   1:L PR[91] R[100]mm/sec CNT100;
   1:  PR[91,1] = PR[90,1] + 41.639;
   1:  PR[91,2] = PR[90,2] + -7.511;
   1:L PR[91] R[100]mm/sec CNT100;
   1:  PR[91,1] = PR[90,1] + 42.015;
   1:  PR[91,2] = PR[90,2] + -6.602;
   1:L PR[91] R[100]mm/sec CNT100;
   1:  PR[91,1] = PR[90,1] + 42.645;
   1:  PR[91,2] = PR[90,2] + -4.250;
   1:L PR[91] R[100]mm/sec CNT100;
   1:  PR[91,1] = PR[90,1] + 42.870;
   1:  PR[91,2] = PR[90,2] + -1.671;
   1:L PR[91] R[100]mm/sec CNT100;
   1:  PR[91,1] = PR[90,1] + 42.984;
   1:  PR[91,2] = PR[90,2] + -0.700;
   1:L PR[91] R[100]mm/sec CNT100;
   1:  PR[91,1] = PR[90,1] + 42.778;
   1:  PR[91,2] = PR[90,2] + 1.658;
   1:L PR[91] R[100]mm/sec CNT100;
   1:  PR[91,1] = PR[90,1] + 42.775;
   1:  PR[91,2] = PR[90,2] + 1.848;
   1:L PR[91] R[100]mm/sec CNT100;
   1:  PR[91,1] = PR[90,1] + 42.656;
   1:  PR[91,2] = PR[90,2] + 2.749;
   1:L PR[91] R[100]mm/sec CNT100;
   1:  PR[91,1] = PR[90,1] + 42.015;
   1:  PR[91,2] = PR[90,2] + 5.145;
   1:L PR[91] R[100]mm/sec CNT100;
   1:  PR[91,1] = PR[90,1] + 41.639;
   1:  PR[91,2] = PR[90,2] + 6.053;
   1:L PR[91] R[100]mm/sec CNT100;
   1:  PR[91,1] = PR[90,1] + 40.576;
   1:  PR[91,2] = PR[90,2] + 8.332;
   1:L PR[91] R[100]mm/sec CNT100;
   1:  PR[91,1] = PR[90,1] + 39.128;
   1:  PR[91,2] = PR[90,2] + 10.399;
   1:L PR[91] R[100]mm/sec CNT100;
   1:  PR[91,1] = PR[90,1] + 38.528;
   1:  PR[91,2] = PR[90,2] + 11.183;
   1:L PR[91] R[100]mm/sec CNT100;
   1:  PR[91,1] = PR[90,1] + 36.785;
   1:  PR[91,2] = PR[90,2] + 12.925;
   1:L PR[91] R[100]mm/sec CNT100;
   1:  PR[91,1] = PR[90,1] + 35.993;
   1:  PR[91,2] = PR[90,2] + 13.534;
   1:L PR[91] R[100]mm/sec CNT100;
   1:  PR[91,1] = PR[90,1] + 33.939;
   1:  PR[91,2] = PR[90,2] + 14.971;
   1:L PR[91] R[100]mm/sec CNT100;
   1:  PR[91,1] = PR[90,1] + 31.670;
   1:  PR[91,2] = PR[90,2] + 16.028;
   1:L PR[91] R[100]mm/sec CNT100;
   1:  PR[91,1] = PR[90,1] + 30.740;
   1:  PR[91,2] = PR[90,2] + 16.415;
   1:L PR[91] R[100]mm/sec CNT100;
   1:  PR[91,1] = PR[90,1] + 28.367;
   1:  PR[91,2] = PR[90,2] + 17.050;
   1:L PR[91] R[100]mm/sec CNT100;
   1:  PR[91,1] = PR[90,1] + 27.353;
   1:  PR[91,2] = PR[90,2] + 17.186;
   1:L PR[91] R[100]mm/sec CNT100;
   1:  PR[91,1] = PR[90,1] + 24.877;
   1:  PR[91,2] = PR[90,2] + 17.401;
   1:L PR[91] R[100]mm/sec CNT100;
   1:  PR[91,1] = PR[90,1] + 22.397;
   1:  PR[91,2] = PR[90,2] + 17.184;
   1:L PR[91] R[100]mm/sec CNT100;
   1:  PR[91,1] = PR[90,1] + 21.373;
   1:  PR[91,2] = PR[90,2] + 17.050;
   1:L PR[91] R[100]mm/sec CNT100;
   1:  PR[91,1] = PR[90,1] + 19.063;
   1:  PR[91,2] = PR[90,2] + 16.431;
   1:L PR[91] R[100]mm/sec CNT100TB   .50sec,CALL END_PUD;
   1:  PR[92] = PR[91];
   1:  PR[92,3] = PR[92,3] + 20;
   1:J PR[92] 10% FINE;
   1:  PR[91,1] = PR[90,1] + 64.674;
   1:  PR[91,2] = PR[90,2] + 14.280;
   1:  PR[92] = PR[91];
   1:  PR[92,3] = PR[92,3] + 20;
   1:J PR[92] 10% FINE;
   1:L PR[91] R[100]mm/sec CNT100;
   1:  CALL LASER_DRAHT_START;
   1:  PR[91,1] = PR[90,1] + 63.262;
   1:  PR[91,2] = PR[90,2] + 13.292;
   1:L PR[91] R[100]mm/sec CNT100;
   1:  PR[91,1] = PR[90,1] + 60.701;
   1:  PR[91,2] = PR[90,2] + 10.743;
   1:L PR[91] R[100]mm/sec CNT100;
   1:  PR[91,1] = PR[90,1] + 59.758;
   1:  PR[91,2] = PR[90,2] + 9.397;
   1:L PR[91] R[100]mm/sec CNT100;
   1:  PR[91,1] = PR[90,1] + 58.704;
   1:  PR[91,2] = PR[90,2] + 7.731;
   1:L PR[91] R[100]mm/sec CNT100;
   1:  PR[91,1] = PR[90,1] + 58.042;
   1:  PR[91,2] = PR[90,2] + 6.310;
   1:L PR[91] R[100]mm/sec CNT100;
   1:  PR[91,1] = PR[90,1] + 57.357;
   1:  PR[91,2] = PR[90,2] + 4.363;
   1:L PR[91] R[100]mm/sec CNT100;
   1:  PR[91,1] = PR[90,1] + 56.969;
   1:  PR[91,2] = PR[90,2] + 2.914;
   1:L PR[91] R[100]mm/sec CNT100;
   1:  PR[91,1] = PR[90,1] + 56.830;
   1:  PR[91,2] = PR[90,2] + 1.324;
   1:L PR[91] R[100]mm/sec CNT100;
   1:  PR[91,1] = PR[90,1] + 56.595;
   1:  PR[91,2] = PR[90,2] + -0.755;
   1:L PR[91] R[100]mm/sec CNT100;
   1:  PR[91,1] = PR[90,1] + 56.725;
   1:  PR[91,2] = PR[90,2] + -2.242;
   1:L PR[91] R[100]mm/sec CNT100;
   1:  PR[91,1] = PR[90,1] + 56.962;
   1:  PR[91,2] = PR[90,2] + -4.348;
   1:L PR[91] R[100]mm/sec CNT100;
   1:  PR[91,1] = PR[90,1] + 57.356;
   1:  PR[91,2] = PR[90,2] + -5.821;
   1:L PR[91] R[100]mm/sec CNT100;
   1:  PR[91,1] = PR[90,1] + 58.041;
   1:  PR[91,2] = PR[90,2] + -7.768;
   1:L PR[91] R[100]mm/sec CNT100;
   1:  PR[91,1] = PR[90,1] + 58.703;
   1:  PR[91,2] = PR[90,2] + -9.188;
   1:L PR[91] R[100]mm/sec CNT100;
   1:  PR[91,1] = PR[90,1] + 59.757;
   1:  PR[91,2] = PR[90,2] + -10.854;
   1:L PR[91] R[100]mm/sec CNT100;
   1:  PR[91,1] = PR[90,1] + 60.699;
   1:  PR[91,2] = PR[90,2] + -12.200;
   1:L PR[91] R[100]mm/sec CNT100;
   1:  PR[91,1] = PR[90,1] + 63.259;
   1:  PR[91,2] = PR[90,2] + -14.749;
   1:L PR[91] R[100]mm/sec CNT100;
   1:  PR[91,1] = PR[90,1] + 64.671;
   1:  PR[91,2] = PR[90,2] + -15.737;
   1:L PR[91] R[100]mm/sec CNT100;
   1:  PR[91,1] = PR[90,1] + 66.191;
   1:  PR[91,2] = PR[90,2] + -16.684;
   1:L PR[91] R[100]mm/sec CNT100;
   1:  PR[91,1] = PR[90,1] + 67.830;
   1:  PR[91,2] = PR[90,2] + -17.448;
   1:L PR[91] R[100]mm/sec CNT100;
   1:  PR[91,1] = PR[90,1] + 69.388;
   1:  PR[91,2] = PR[90,2] + -17.986;
   1:L PR[91] R[100]mm/sec CNT100;
   1:  PR[91,1] = PR[90,1] + 71.205;
   1:  PR[91,2] = PR[90,2] + -18.473;
   1:L PR[91] R[100]mm/sec CNT100;
   1:  PR[91,1] = PR[90,1] + 73.166;
   1:  PR[91,2] = PR[90,2] + -18.646;
   1:L PR[91] R[100]mm/sec CNT100;
   1:  PR[91,1] = PR[90,1] + 74.752;
   1:  PR[91,2] = PR[90,2] + -18.816;
   1:L PR[91] R[100]mm/sec CNT100;
   1:  PR[91,1] = PR[90,1] + 76.727;
   1:  PR[91,2] = PR[90,2] + -18.644;
   1:L PR[91] R[100]mm/sec CNT100;
   1:  PR[91,1] = PR[90,1] + 78.184;
   1:  PR[91,2] = PR[90,2] + -18.473;
   1:L PR[91] R[100]mm/sec CNT100;
   1:  PR[91,1] = PR[90,1] + 80.174;
   1:  PR[91,2] = PR[90,2] + -17.941;
   1:L PR[91] R[100]mm/sec CNT100;
   1:  PR[91,1] = PR[90,1] + 81.453;
   1:  PR[91,2] = PR[90,2] + -17.489;
   1:L PR[91] R[100]mm/sec CNT100;
   1:  PR[91,1] = PR[90,1] + 83.371;
   1:  PR[91,2] = PR[90,2] + -16.595;
   1:L PR[91] R[100]mm/sec CNT100;
   1:  PR[91,1] = PR[90,1] + 84.442;
   1:  PR[91,2] = PR[90,2] + -15.917;
   1:L PR[91] R[100]mm/sec CNT100;
   1:  PR[91,1] = PR[90,1] + 86.225;
   1:  PR[91,2] = PR[90,2] + -14.670;
   1:L PR[91] R[100]mm/sec CNT100;
   1:  PR[91,1] = PR[90,1] + 87.789;
   1:  PR[91,2] = PR[90,2] + -13.107;
   1:L PR[91] R[100]mm/sec CNT100;
   1:  PR[91,1] = PR[90,1] + 88.663;
   1:  PR[91,2] = PR[90,2] + -12.228;
   1:L PR[91] R[100]mm/sec CNT100;
   1:  PR[91,1] = PR[90,1] + 89.933;
   1:  PR[91,2] = PR[90,2] + -10.414;
   1:L PR[91] R[100]mm/sec CNT100;
   1:  PR[91,1] = PR[90,1] + 90.561;
   1:  PR[91,2] = PR[90,2] + -9.412;
   1:L PR[91] R[100]mm/sec CNT100;
   1:  PR[91,1] = PR[90,1] + 91.506;
   1:  PR[91,2] = PR[90,2] + -7.386;
   1:L PR[91] R[100]mm/sec CNT100;
   1:  PR[91,1] = PR[90,1] + 91.883;
   1:  PR[91,2] = PR[90,2] + -6.304;
   1:L PR[91] R[100]mm/sec CNT100;
   1:  PR[91,1] = PR[90,1] + 92.460;
   1:  PR[91,2] = PR[90,2] + -4.148;
   1:L PR[91] R[100]mm/sec CNT100;
   1:  PR[91,1] = PR[90,1] + 92.662;
   1:  PR[91,2] = PR[90,2] + -1.835;
   1:L PR[91] R[100]mm/sec CNT100;
   1:  PR[91,1] = PR[90,1] + 92.788;
   1:  PR[91,2] = PR[90,2] + -0.706;
   1:L PR[91] R[100]mm/sec CNT100;
   1:  PR[91,1] = PR[90,1] + 92.590;
   1:  PR[91,2] = PR[90,2] + 1.557;
   1:L PR[91] R[100]mm/sec CNT100;
   1:  PR[91,1] = PR[90,1] + 92.466;
   1:  PR[91,2] = PR[90,2] + 2.666;
   1:L PR[91] R[100]mm/sec CNT100;
   1:  PR[91,1] = PR[90,1] + 91.883;
   1:  PR[91,2] = PR[90,2] + 4.844;
   1:L PR[91] R[100]mm/sec CNT100;
   1:  PR[91,1] = PR[90,1] + 91.506;
   1:  PR[91,2] = PR[90,2] + 5.927;
   1:L PR[91] R[100]mm/sec CNT100;
   1:  PR[91,1] = PR[90,1] + 90.562;
   1:  PR[91,2] = PR[90,2] + 7.951;
   1:L PR[91] R[100]mm/sec CNT100;
   1:  PR[91,1] = PR[90,1] + 89.935;
   1:  PR[91,2] = PR[90,2] + 8.953;
   1:L PR[91] R[100]mm/sec CNT100;
   1:  PR[91,1] = PR[90,1] + 88.666;
   1:  PR[91,2] = PR[90,2] + 10.765;
   1:L PR[91] R[100]mm/sec CNT100;
   1:  PR[91,1] = PR[90,1] + 86.227;
   1:  PR[91,2] = PR[90,2] + 13.209;
   1:L PR[91] R[100]mm/sec CNT100;
   1:  PR[91,1] = PR[90,1] + 84.447;
   1:  PR[91,2] = PR[90,2] + 14.456;
   1:L PR[91] R[100]mm/sec CNT100;
   1:  PR[91,1] = PR[90,1] + 83.376;
   1:  PR[91,2] = PR[90,2] + 15.134;
   1:L PR[91] R[100]mm/sec CNT100;
   1:  PR[91,1] = PR[90,1] + 81.460;
   1:  PR[91,2] = PR[90,2] + 16.027;
   1:L PR[91] R[100]mm/sec CNT100;
   1:  PR[91,1] = PR[90,1] + 80.180;
   1:  PR[91,2] = PR[90,2] + 16.480;
   1:L PR[91] R[100]mm/sec CNT100;
   1:  PR[91,1] = PR[90,1] + 78.221;
   1:  PR[91,2] = PR[90,2] + 17.005;
   1:L PR[91] R[100]mm/sec CNT100;
   1:  PR[91,1] = PR[90,1] + 76.094;
   1:  PR[91,2] = PR[90,2] + 17.192;
   1:L PR[91] R[100]mm/sec CNT100;
   1:  PR[91,1] = PR[90,1] + 74.710;
   1:  PR[91,2] = PR[90,2] + 17.356;
   1:L PR[91] R[100]mm/sec CNT100;
   1:  PR[91,1] = PR[90,1] + 72.737;
   1:  PR[91,2] = PR[90,2] + 17.184;
   1:L PR[91] R[100]mm/sec CNT100;
   1:  PR[91,1] = PR[90,1] + 71.232;
   1:  PR[91,2] = PR[90,2] + 17.021;
   1:L PR[91] R[100]mm/sec CNT100;
   1:  PR[91,1] = PR[90,1] + 69.394;
   1:  PR[91,2] = PR[90,2] + 16.530;
   1:L PR[91] R[100]mm/sec CNT100;
   1:  PR[91,1] = PR[90,1] + 67.835;
   1:  PR[91,2] = PR[90,2] + 15.992;
   1:L PR[91] R[100]mm/sec CNT100;
   1:  PR[91,1] = PR[90,1] + 66.195;
   1:  PR[91,2] = PR[90,2] + 15.227;
   1:L PR[91] R[100]mm/sec CNT100;
   1:  PR[91,1] = PR[90,1] + 64.674;
   1:  PR[91,2] = PR[90,2] + 14.280;
   1:L PR[91] R[100]mm/sec CNT100TB   .50sec,CALL END_PUD;
   1:  PR[92] = PR[91];
   1:  PR[92,3] = PR[92,3] + 20;
   1:J PR[92] 10% FINE;
   1:  PR[91,1] = PR[90,1] + -7.150;
   1:  PR[91,2] = PR[90,2] + 2.703;
   1:  PR[92] = PR[91];
   1:  PR[92,3] = PR[92,3] + 20;
   1:J PR[92] 10% FINE;
   1:L PR[91] R[100]mm/sec CNT100;
   1:  CALL LASER_DRAHT_START;
   1:  PR[91,1] = PR[90,1] + -7.705;
   1:  PR[91,2] = PR[90,2] + 4.775;
   1:L PR[91] R[100]mm/sec CNT100;
   1:  PR[91,1] = PR[90,1] + -8.126;
   1:  PR[91,2] = PR[90,2] + 5.975;
   1:L PR[91] R[100]mm/sec CNT100;
   1:  PR[91,1] = PR[90,1] + -9.039;
   1:  PR[91,2] = PR[90,2] + 7.935;
   1:L PR[91] R[100]mm/sec CNT100;
   1:  PR[91,1] = PR[90,1] + -9.701;
   1:  PR[91,2] = PR[90,2] + 8.983;
   1:L PR[91] R[100]mm/sec CNT100;
   1:  PR[91,1] = PR[90,1] + -10.954;
   1:  PR[91,2] = PR[90,2] + 10.774;
   1:L PR[91] R[100]mm/sec CNT100;
   1:  PR[91,1] = PR[90,1] + -13.403;
   1:  PR[91,2] = PR[90,2] + 13.218;
   1:L PR[91] R[100]mm/sec CNT100;
   1:  PR[91,1] = PR[90,1] + -15.216;
   1:  PR[91,2] = PR[90,2] + 14.488;
   1:L PR[91] R[100]mm/sec CNT100;
   1:  PR[91,1] = PR[90,1] + -16.211;
   1:  PR[91,2] = PR[90,2] + 15.110;
   1:L PR[91] R[100]mm/sec CNT100;
   1:  PR[91,1] = PR[90,1] + -18.252;
   1:  PR[91,2] = PR[90,2] + 16.062;
   1:L PR[91] R[100]mm/sec CNT100;
   1:  PR[91,1] = PR[90,1] + -19.306;
   1:  PR[91,2] = PR[90,2] + 16.427;
   1:L PR[91] R[100]mm/sec CNT100;
   1:  PR[91,1] = PR[90,1] + -21.495;
   1:  PR[91,2] = PR[90,2] + 17.014;
   1:L PR[91] R[100]mm/sec CNT100;
   1:  PR[91,1] = PR[90,1] + -23.847;
   1:  PR[91,2] = PR[90,2] + 17.220;
   1:L PR[91] R[100]mm/sec CNT100;
   1:  PR[91,1] = PR[90,1] + -24.934;
   1:  PR[91,2] = PR[90,2] + 17.339;
   1:L PR[91] R[100]mm/sec CNT100;
   1:  PR[91,1] = PR[90,1] + -27.250;
   1:  PR[91,2] = PR[90,2] + 17.136;
   1:L PR[91] R[100]mm/sec CNT100;
   1:  PR[91,1] = PR[90,1] + -28.281;
   1:  PR[91,2] = PR[90,2] + 17.016;
   1:L PR[91] R[100]mm/sec CNT100;
   1:  PR[91,1] = PR[90,1] + -30.558;
   1:  PR[91,2] = PR[90,2] + 16.406;
   1:L PR[91] R[100]mm/sec CNT100;
   1:  PR[91,1] = PR[90,1] + -31.489;
   1:  PR[91,2] = PR[90,2] + 16.077;
   1:L PR[91] R[100]mm/sec CNT100;
   1:  PR[91,1] = PR[90,1] + -33.652;
   1:  PR[91,2] = PR[90,2] + 15.068;
   1:L PR[91] R[100]mm/sec CNT100;
   1:  PR[91,1] = PR[90,1] + -34.450;
   1:  PR[91,2] = PR[90,2] + 14.564;
   1:L PR[91] R[100]mm/sec CNT100;
   1:  PR[91,1] = PR[90,1] + -36.424;
   1:  PR[91,2] = PR[90,2] + 13.181;
   1:L PR[91] R[100]mm/sec CNT100;
   1:  PR[91,1] = PR[90,1] + -38.821;
   1:  PR[91,2] = PR[90,2] + 10.781;
   1:L PR[91] R[100]mm/sec CNT100;
   1:  PR[91,1] = PR[90,1] + -40.213;
   1:  PR[91,2] = PR[90,2] + 8.792;
   1:L PR[91] R[100]mm/sec CNT100;
   1:  PR[91,1] = PR[90,1] + -40.692;
   1:  PR[91,2] = PR[90,2] + 8.028;
   1:L PR[91] R[100]mm/sec CNT100;
   1:  PR[91,1] = PR[90,1] + -41.725;
   1:  PR[91,2] = PR[90,2] + 5.811;
   1:L PR[91] R[100]mm/sec CNT100;
   1:  PR[91,1] = PR[90,1] + -42.016;
   1:  PR[91,2] = PR[90,2] + 4.978;
   1:L PR[91] R[100]mm/sec CNT100;
   1:  PR[91,1] = PR[90,1] + -42.644;
   1:  PR[91,2] = PR[90,2] + 2.633;
   1:L PR[91] R[100]mm/sec CNT100;
   1:  PR[91,1] = PR[90,1] + -42.864;
   1:  PR[91,2] = PR[90,2] + 0.118;
   1:L PR[91] R[100]mm/sec CNT100;
   1:  PR[91,1] = PR[90,1] + -42.962;
   1:  PR[91,2] = PR[90,2] + -0.754;
   1:L PR[91] R[100]mm/sec CNT100;
   1:  PR[91,1] = PR[90,1] + -42.748;
   1:  PR[91,2] = PR[90,2] + -3.198;
   1:L PR[91] R[100]mm/sec CNT100;
   1:  PR[91,1] = PR[90,1] + -42.650;
   1:  PR[91,2] = PR[90,2] + -4.066;
   1:L PR[91] R[100]mm/sec CNT100;
   1:  PR[91,1] = PR[90,1] + -42.016;
   1:  PR[91,2] = PR[90,2] + -6.436;
   1:L PR[91] R[100]mm/sec CNT100;
   1:  PR[91,1] = PR[90,1] + -41.725;
   1:  PR[91,2] = PR[90,2] + -7.269;
   1:L PR[91] R[100]mm/sec CNT100;
   1:  PR[91,1] = PR[90,1] + -40.692;
   1:  PR[91,2] = PR[90,2] + -9.486;
   1:L PR[91] R[100]mm/sec CNT100;
   1:  PR[91,1] = PR[90,1] + -40.214;
   1:  PR[91,2] = PR[90,2] + -10.250;
   1:L PR[91] R[100]mm/sec CNT100;
   1:  PR[91,1] = PR[90,1] + -38.822;
   1:  PR[91,2] = PR[90,2] + -12.239;
   1:L PR[91] R[100]mm/sec CNT100;
   1:  PR[91,1] = PR[90,1] + -36.425;
   1:  PR[91,2] = PR[90,2] + -14.639;
   1:L PR[91] R[100]mm/sec CNT100;
   1:  PR[91,1] = PR[90,1] + -34.451;
   1:  PR[91,2] = PR[90,2] + -16.022;
   1:L PR[91] R[100]mm/sec CNT100;
   1:  PR[91,1] = PR[90,1] + -33.653;
   1:  PR[91,2] = PR[90,2] + -16.527;
   1:L PR[91] R[100]mm/sec CNT100;
   1:  PR[91,1] = PR[90,1] + -31.490;
   1:  PR[91,2] = PR[90,2] + -17.536;
   1:L PR[91] R[100]mm/sec CNT100;
   1:  PR[91,1] = PR[90,1] + -30.559;
   1:  PR[91,2] = PR[90,2] + -17.864;
   1:L PR[91] R[100]mm/sec CNT100;
   1:  PR[91,1] = PR[90,1] + -28.309;
   1:  PR[91,2] = PR[90,2] + -18.467;
   1:L PR[91] R[100]mm/sec CNT100;
   1:  PR[91,1] = PR[90,1] + -25.882;
   1:  PR[91,2] = PR[90,2] + -18.680;
   1:L PR[91] R[100]mm/sec CNT100;
   1:  PR[91,1] = PR[90,1] + -24.884;
   1:  PR[91,2] = PR[90,2] + -18.797;
   1:L PR[91] R[100]mm/sec CNT100;
   1:  PR[91,1] = PR[90,1] + -22.569;
   1:  PR[91,2] = PR[90,2] + -18.594;
   1:L PR[91] R[100]mm/sec CNT100;
   1:  PR[91,1] = PR[90,1] + -21.517;
   1:  PR[91,2] = PR[90,2] + -18.479;
   1:L PR[91] R[100]mm/sec CNT100;
   1:  PR[91,1] = PR[90,1] + -19.307;
   1:  PR[91,2] = PR[90,2] + -17.886;
   1:L PR[91] R[100]mm/sec CNT100;
   1:  PR[91,1] = PR[90,1] + -18.253;
   1:  PR[91,2] = PR[90,2] + -17.521;
   1:L PR[91] R[100]mm/sec CNT100;
   1:  PR[91,1] = PR[90,1] + -16.212;
   1:  PR[91,2] = PR[90,2] + -16.569;
   1:L PR[91] R[100]mm/sec CNT100;
   1:  PR[91,1] = PR[90,1] + -15.217;
   1:  PR[91,2] = PR[90,2] + -15.948;
   1:L PR[91] R[100]mm/sec CNT100;
   1:  PR[91,1] = PR[90,1] + -13.404;
   1:  PR[91,2] = PR[90,2] + -14.678;
   1:L PR[91] R[100]mm/sec CNT100;
   1:  PR[91,1] = PR[90,1] + -10.955;
   1:  PR[91,2] = PR[90,2] + -12.233;
   1:L PR[91] R[100]mm/sec CNT100;
   1:  PR[91,1] = PR[90,1] + -9.702;
   1:  PR[91,2] = PR[90,2] + -10.443;
   1:L PR[91] R[100]mm/sec CNT100;
   1:  PR[91,1] = PR[90,1] + -9.040;
   1:  PR[91,2] = PR[90,2] + -9.394;
   1:L PR[91] R[100]mm/sec CNT100;
   1:  PR[91,1] = PR[90,1] + -8.127;
   1:  PR[91,2] = PR[90,2] + -7.435;
   1:L PR[91] R[100]mm/sec CNT100;
   1:  PR[91,1] = PR[90,1] + -7.705;
   1:  PR[91,2] = PR[90,2] + -6.234;
   1:L PR[91] R[100]mm/sec CNT100;
   1:  PR[91,1] = PR[90,1] + -7.157;
   1:  PR[91,2] = PR[90,2] + -4.187;
   1:L PR[91] R[100]mm/sec CNT100;
   1:  PR[91,1] = PR[90,1] + -6.965;
   1:  PR[91,2] = PR[90,2] + -1.986;
   1:L PR[91] R[100]mm/sec CNT100;
   1:  PR[91,1] = PR[90,1] + -6.832;
   1:  PR[91,2] = PR[90,2] + -0.713;
   1:L PR[91] R[100]mm/sec CNT100;
   1:  PR[91,1] = PR[90,1] + -7.035;
   1:  PR[91,2] = PR[90,2] + 1.604;
   1:L PR[91] R[100]mm/sec CNT100;
   1:  PR[91,1] = PR[90,1] + -7.030;
   1:  PR[91,2] = PR[90,2] + 1.640;
   1:L PR[91] R[100]mm/sec CNT100;
   1:  PR[91,1] = PR[90,1] + -7.150;
   1:  PR[91,2] = PR[90,2] + 2.703;
   1:L PR[91] R[100]mm/sec CNT100TB   .50sec,CALL END_PUD;
   1:  PR[92] = PR[91];
   1:  PR[92,3] = PR[92,3] + 20;
   1:J PR[92] 10% FINE;
   1:  PR[91,1] = PR[90,1] + -92.606;
   1:  PR[91,2] = PR[90,2] + 2.602;
   1:  PR[92] = PR[91];
   1:  PR[92,3] = PR[92,3] + 20;
   1:J PR[92] 10% FINE;
   1:L PR[91] R[100]mm/sec CNT100;
   1:  CALL LASER_DRAHT_START;
   1:  PR[91,1] = PR[90,1] + -92.805;
   1:  PR[91,2] = PR[90,2] + 0.315;
   1:L PR[91] R[100]mm/sec CNT100;
   1:  PR[91,1] = PR[90,1] + -92.917;
   1:  PR[91,2] = PR[90,2] + -0.747;
   1:L PR[91] R[100]mm/sec CNT100;
   1:  PR[91,1] = PR[90,1] + -92.733;
   1:  PR[91,2] = PR[90,2] + -2.852;
   1:L PR[91] R[100]mm/sec CNT100;
   1:  PR[91,1] = PR[90,1] + -92.712;
   1:  PR[91,2] = PR[90,2] + -2.937;
   1:L PR[91] R[100]mm/sec CNT100;
   1:  PR[91,1] = PR[90,1] + -92.598;
   1:  PR[91,2] = PR[90,2] + -4.024;
   1:L PR[91] R[100]mm/sec CNT100;
   1:  PR[91,1] = PR[90,1] + -91.988;
   1:  PR[91,2] = PR[90,2] + -6.299;
   1:L PR[91] R[100]mm/sec CNT100;
   1:  PR[91,1] = PR[90,1] + -91.696;
   1:  PR[91,2] = PR[90,2] + -7.202;
   1:L PR[91] R[100]mm/sec CNT100;
   1:  PR[91,1] = PR[90,1] + -90.708;
   1:  PR[91,2] = PR[90,2] + -9.320;
   1:L PR[91] R[100]mm/sec CNT100;
   1:  PR[91,1] = PR[90,1] + -90.223;
   1:  PR[91,2] = PR[90,2] + -10.162;
   1:L PR[91] R[100]mm/sec CNT100;
   1:  PR[91,1] = PR[90,1] + -88.889;
   1:  PR[91,2] = PR[90,2] + -12.065;
   1:L PR[91] R[100]mm/sec CNT100;
   1:  PR[91,1] = PR[90,1] + -88.216;
   1:  PR[91,2] = PR[90,2] + -12.815;
   1:L PR[91] R[100]mm/sec CNT100;
   1:  PR[91,1] = PR[90,1] + -86.600;
   1:  PR[91,2] = PR[90,2] + -14.431;
   1:L PR[91] R[100]mm/sec CNT100;
   1:  PR[91,1] = PR[90,1] + -85.745;
   1:  PR[91,2] = PR[90,2] + -15.054;
   1:L PR[91] R[100]mm/sec CNT100;
   1:  PR[91,1] = PR[90,1] + -83.886;
   1:  PR[91,2] = PR[90,2] + -16.355;
   1:L PR[91] R[100]mm/sec CNT100;
   1:  PR[91,1] = PR[90,1] + -81.830;
   1:  PR[91,2] = PR[90,2] + -17.313;
   1:L PR[91] R[100]mm/sec CNT100;
   1:  PR[91,1] = PR[90,1] + -80.849;
   1:  PR[91,2] = PR[90,2] + -17.752;
   1:L PR[91] R[100]mm/sec CNT100;
   1:  PR[91,1] = PR[90,1] + -78.718;
   1:  PR[91,2] = PR[90,2] + -18.322;
   1:L PR[91] R[100]mm/sec CNT100;
   1:  PR[91,1] = PR[90,1] + -77.600;
   1:  PR[91,2] = PR[90,2] + -18.562;
   1:L PR[91] R[100]mm/sec CNT100;
   1:  PR[91,1] = PR[90,1] + -75.458;
   1:  PR[91,2] = PR[90,2] + -18.749;
   1:L PR[91] R[100]mm/sec CNT100;
   1:  PR[91,1] = PR[90,1] + -74.234;
   1:  PR[91,2] = PR[90,2] + -18.752;
   1:L PR[91] R[100]mm/sec CNT100;
   1:  PR[91,1] = PR[90,1] + -72.153;
   1:  PR[91,2] = PR[90,2] + -18.569;
   1:L PR[91] R[100]mm/sec CNT100;
   1:  PR[91,1] = PR[90,1] + -70.867;
   1:  PR[91,2] = PR[90,2] + -18.299;
   1:L PR[91] R[100]mm/sec CNT100;
   1:  PR[91,1] = PR[90,1] + -68.931;
   1:  PR[91,2] = PR[90,2] + -17.780;
   1:L PR[91] R[100]mm/sec CNT100;
   1:  PR[91,1] = PR[90,1] + -67.051;
   1:  PR[91,2] = PR[90,2] + -16.902;
   1:L PR[91] R[100]mm/sec CNT100;
   1:  PR[91,1] = PR[90,1] + -65.823;
   1:  PR[91,2] = PR[90,2] + -16.361;
   1:L PR[91] R[100]mm/sec CNT100;
   1:  PR[91,1] = PR[90,1] + -64.221;
   1:  PR[91,2] = PR[90,2] + -15.239;
   1:L PR[91] R[100]mm/sec CNT100;
   1:  PR[91,1] = PR[90,1] + -63.053;
   1:  PR[91,2] = PR[90,2] + -14.396;
   1:L PR[91] R[100]mm/sec CNT100;
   1:  PR[91,1] = PR[90,1] + -61.723;
   1:  PR[91,2] = PR[90,2] + -13.066;
   1:L PR[91] R[100]mm/sec CNT100;
   1:  PR[91,1] = PR[90,1] + -60.695;
   1:  PR[91,2] = PR[90,2] + -11.928;
   1:L PR[91] R[100]mm/sec CNT100;
   1:  PR[91,1] = PR[90,1] + -59.646;
   1:  PR[91,2] = PR[90,2] + -10.430;
   1:L PR[91] R[100]mm/sec CNT100;
   1:  PR[91,1] = PR[90,1] + -58.837;
   1:  PR[91,2] = PR[90,2] + -9.034;
   1:L PR[91] R[100]mm/sec CNT100;
   1:  PR[91,1] = PR[90,1] + -58.088;
   1:  PR[91,2] = PR[90,2] + -7.427;
   1:L PR[91] R[100]mm/sec CNT100;
   1:  PR[91,1] = PR[90,1] + -57.571;
   1:  PR[91,2] = PR[90,2] + -5.839;
   1:L PR[91] R[100]mm/sec CNT100;
   1:  PR[91,1] = PR[90,1] + -57.124;
   1:  PR[91,2] = PR[90,2] + -4.170;
   1:L PR[91] R[100]mm/sec CNT100;
   1:  PR[91,1] = PR[90,1] + -56.818;
   1:  PR[91,2] = PR[90,2] + -0.728;
   1:L PR[91] R[100]mm/sec CNT100;
   1:  PR[91,1] = PR[90,1] + -56.955;
   1:  PR[91,2] = PR[90,2] + 0.839;
   1:L PR[91] R[100]mm/sec CNT100;
   1:  PR[91,1] = PR[90,1] + -57.154;
   1:  PR[91,2] = PR[90,2] + 2.727;
   1:L PR[91] R[100]mm/sec CNT100;
   1:  PR[91,1] = PR[90,1] + -57.562;
   1:  PR[91,2] = PR[90,2] + 4.249;
   1:L PR[91] R[100]mm/sec CNT100;
   1:  PR[91,1] = PR[90,1] + -58.141;
   1:  PR[91,2] = PR[90,2] + 6.028;
   1:L PR[91] R[100]mm/sec CNT100;
   1:  PR[91,1] = PR[90,1] + -58.820;
   1:  PR[91,2] = PR[90,2] + 7.485;
   1:L PR[91] R[100]mm/sec CNT100;
   1:  PR[91,1] = PR[90,1] + -59.727;
   1:  PR[91,2] = PR[90,2] + 9.050;
   1:L PR[91] R[100]mm/sec CNT100;
   1:  PR[91,1] = PR[90,1] + -60.684;
   1:  PR[91,2] = PR[90,2] + 10.416;
   1:L PR[91] R[100]mm/sec CNT100;
   1:  PR[91,1] = PR[90,1] + -61.836;
   1:  PR[91,2] = PR[90,2] + 11.693;
   1:L PR[91] R[100]mm/sec CNT100;
   1:  PR[91,1] = PR[90,1] + -63.059;
   1:  PR[91,2] = PR[90,2] + 12.914;
   1:L PR[91] R[100]mm/sec CNT100;
   1:  PR[91,1] = PR[90,1] + -64.369;
   1:  PR[91,2] = PR[90,2] + 13.862;
   1:L PR[91] R[100]mm/sec CNT100;
   1:  PR[91,1] = PR[90,1] + -65.867;
   1:  PR[91,2] = PR[90,2] + 14.910;
   1:L PR[91] R[100]mm/sec CNT100;
   1:  PR[91,1] = PR[90,1] + -67.518;
   1:  PR[91,2] = PR[90,2] + 15.679;
   1:L PR[91] R[100]mm/sec CNT100;
   1:  PR[91,1] = PR[90,1] + -68.967;
   1:  PR[91,2] = PR[90,2] + 16.321;
   1:L PR[91] R[100]mm/sec CNT100;
   1:  PR[91,1] = PR[90,1] + -70.788;
   1:  PR[91,2] = PR[90,2] + 16.808;
   1:L PR[91] R[100]mm/sec CNT100;
   1:  PR[91,1] = PR[90,1] + -72.235;
   1:  PR[91,2] = PR[90,2] + 17.113;
   1:L PR[91] R[100]mm/sec CNT100;
   1:  PR[91,1] = PR[90,1] + -74.185;
   1:  PR[91,2] = PR[90,2] + 17.283;
   1:L PR[91] R[100]mm/sec CNT100;
   1:  PR[91,1] = PR[90,1] + -75.563;
   1:  PR[91,2] = PR[90,2] + 17.281;
   1:L PR[91] R[100]mm/sec CNT100;
   1:  PR[91,1] = PR[90,1] + -77.579;
   1:  PR[91,2] = PR[90,2] + 17.104;
   1:L PR[91] R[100]mm/sec CNT100;
   1:  PR[91,1] = PR[90,1] + -78.839;
   1:  PR[91,2] = PR[90,2] + 16.834;
   1:L PR[91] R[100]mm/sec CNT100;
   1:  PR[91,1] = PR[90,1] + -80.837;
   1:  PR[91,2] = PR[90,2] + 16.298;
   1:L PR[91] R[100]mm/sec CNT100;
   1:  PR[91,1] = PR[90,1] + -82.768;
   1:  PR[91,2] = PR[90,2] + 15.397;
   1:L PR[91] R[100]mm/sec CNT100;
   1:  PR[91,1] = PR[90,1] + -83.921;
   1:  PR[91,2] = PR[90,2] + 14.881;
   1:L PR[91] R[100]mm/sec CNT100;
   1:  PR[91,1] = PR[90,1] + -85.673;
   1:  PR[91,2] = PR[90,2] + 13.654;
   1:L PR[91] R[100]mm/sec CNT100;
   1:  PR[91,1] = PR[90,1] + -86.638;
   1:  PR[91,2] = PR[90,2] + 12.951;
   1:L PR[91] R[100]mm/sec CNT100;
   1:  PR[91,1] = PR[90,1] + -88.175;
   1:  PR[91,2] = PR[90,2] + 11.414;
   1:L PR[91] R[100]mm/sec CNT100;
   1:  PR[91,1] = PR[90,1] + -88.935;
   1:  PR[91,2] = PR[90,2] + 10.567;
   1:L PR[91] R[100]mm/sec CNT100;
   1:  PR[91,1] = PR[90,1] + -90.206;
   1:  PR[91,2] = PR[90,2] + 8.752;
   1:L PR[91] R[100]mm/sec CNT100;
   1:  PR[91,1] = PR[90,1] + -90.755;
   1:  PR[91,2] = PR[90,2] + 7.801;
   1:L PR[91] R[100]mm/sec CNT100;
   1:  PR[91,1] = PR[90,1] + -91.697;
   1:  PR[91,2] = PR[90,2] + 5.779;
   1:L PR[91] R[100]mm/sec CNT100;
   1:  PR[91,1] = PR[90,1] + -92.028;
   1:  PR[91,2] = PR[90,2] + 4.758;
   1:L PR[91] R[100]mm/sec CNT100;
   1:  PR[91,1] = PR[90,1] + -92.606;
   1:  PR[91,2] = PR[90,2] + 2.602;
   1:L PR[91] R[100]mm/sec CNT100TB   .50sec,CALL END_PUD;
   1:  PR[92] = PR[91];
   1:  PR[92,3] = PR[92,3] + 20;
   1:J PR[92] 10% FINE;
   1:  PR[91] = PR[90];
   1:  PR[91,1] = PR[90,1] + 41.538;
   1:  PR[91,2] = PR[90,2] + 6.352;
   1:  PR[91,3] = PR[90,3] + 13.195;
   1:  PR[92] = PR[91];
   1:  PR[92,3] = PR[92,3] + 20;
   1:J PR[92] 10% FINE;
   1:L PR[91] R[100]mm/sec CNT100;
   1:  CALL LASER_DRAHT_START;
   1:  PR[91,1] = PR[90,1] + 40.602;
   1:  PR[91,2] = PR[90,2] + 8.358;
   1:L PR[91] R[100]mm/sec CNT100;
   1:  PR[91,1] = PR[90,1] + 39.328;
   1:  PR[91,2] = PR[90,2] + 10.178;
   1:L PR[91] R[100]mm/sec CNT100;
   1:  PR[91,1] = PR[90,1] + 38.444;
   1:  PR[91,2] = PR[90,2] + 11.332;
   1:L PR[91] R[100]mm/sec CNT100;
   1:  PR[91,1] = PR[90,1] + 36.915;
   1:  PR[91,2] = PR[90,2] + 12.859;
   1:L PR[91] R[100]mm/sec CNT100;
   1:  PR[91,1] = PR[90,1] + 35.751;
   1:  PR[91,2] = PR[90,2] + 13.755;
   1:L PR[91] R[100]mm/sec CNT100;
   1:  PR[91,1] = PR[90,1] + 33.947;
   1:  PR[91,2] = PR[90,2] + 15.017;
   1:L PR[91] R[100]mm/sec CNT100;
   1:  PR[91,1] = PR[90,1] + 31.954;
   1:  PR[91,2] = PR[90,2] + 15.946;
   1:L PR[91] R[100]mm/sec CNT100;
   1:  PR[91,1] = PR[90,1] + 30.588;
   1:  PR[91,2] = PR[90,2] + 16.514;
   1:L PR[91] R[100]mm/sec CNT100;
   1:  PR[91,1] = PR[90,1] + 28.514;
   1:  PR[91,2] = PR[90,2] + 17.069;
   1:L PR[91] R[100]mm/sec CNT100;
   1:  PR[91,1] = PR[90,1] + 27.024;
   1:  PR[91,2] = PR[90,2] + 17.268;
   1:L PR[91] R[100]mm/sec CNT100;
   1:  PR[91,1] = PR[90,1] + 24.858;
   1:  PR[91,2] = PR[90,2] + 17.457;
   1:L PR[91] R[100]mm/sec CNT100;
   1:  PR[91,1] = PR[90,1] + 22.689;
   1:  PR[91,2] = PR[90,2] + 17.266;
   1:L PR[91] R[100]mm/sec CNT100;
   1:  PR[91,1] = PR[90,1] + 21.186;
   1:  PR[91,2] = PR[90,2] + 17.071;
   1:L PR[91] R[100]mm/sec CNT100;
   1:  PR[91,1] = PR[90,1] + 19.181;
   1:  PR[91,2] = PR[90,2] + 16.533;
   1:L PR[91] R[100]mm/sec CNT100;
   1:  PR[91,1] = PR[90,1] + 17.142;
   1:  PR[91,2] = PR[90,2] + 15.582;
   1:L PR[91] R[100]mm/sec CNT100;
   1:  PR[91,1] = PR[90,1] + 15.729;
   1:  PR[91,2] = PR[90,2] + 15.000;
   1:L PR[91] R[100]mm/sec CNT100;
   1:  PR[91,1] = PR[90,1] + 14.000;
   1:  PR[91,2] = PR[90,2] + 13.789;
   1:L PR[91] R[100]mm/sec CNT100;
   1:  PR[91,1] = PR[90,1] + 12.767;
   1:  PR[91,2] = PR[90,2] + 12.846;
   1:L PR[91] R[100]mm/sec CNT100;
   1:  PR[91,1] = PR[90,1] + 11.286;
   1:  PR[91,2] = PR[90,2] + 11.364;
   1:L PR[91] R[100]mm/sec CNT100;
   1:  PR[91,1] = PR[90,1] + 10.329;
   1:  PR[91,2] = PR[90,2] + 10.119;
   1:L PR[91] R[100]mm/sec CNT100;
   1:  PR[91,1] = PR[90,1] + 9.102;
   1:  PR[91,2] = PR[90,2] + 8.367;
   1:L PR[91] R[100]mm/sec CNT100;
   1:  PR[91,1] = PR[90,1] + 8.200;
   1:  PR[91,2] = PR[90,2] + 6.433;
   1:L PR[91] R[100]mm/sec CNT100;
   1:  PR[91,1] = PR[90,1] + 7.596;
   1:  PR[91,2] = PR[90,2] + 4.977;
   1:L PR[91] R[100]mm/sec CNT100;
   1:  PR[91,1] = PR[90,1] + 7.067;
   1:  PR[91,2] = PR[90,2] + 3.001;
   1:L PR[91] R[100]mm/sec CNT100;
   1:  PR[91,1] = PR[90,1] + 6.874;
   1:  PR[91,2] = PR[90,2] + 0.796;
   1:L PR[91] R[100]mm/sec CNT100;
   1:  PR[91,1] = PR[90,1] + 6.670;
   1:  PR[91,2] = PR[90,2] + -0.772;
   1:L PR[91] R[100]mm/sec CNT100;
   1:  PR[91,1] = PR[90,1] + 6.857;
   1:  PR[91,2] = PR[90,2] + -2.916;
   1:L PR[91] R[100]mm/sec CNT100;
   1:  PR[91,1] = PR[90,1] + 7.055;
   1:  PR[91,2] = PR[90,2] + -4.417;
   1:L PR[91] R[100]mm/sec CNT100;
   1:  PR[91,1] = PR[90,1] + 7.596;
   1:  PR[91,2] = PR[90,2] + -6.437;
   1:L PR[91] R[100]mm/sec CNT100;
   1:  PR[91,1] = PR[90,1] + 8.200;
   1:  PR[91,2] = PR[90,2] + -7.893;
   1:L PR[91] R[100]mm/sec CNT100;
   1:  PR[91,1] = PR[90,1] + 9.103;
   1:  PR[91,2] = PR[90,2] + -9.828;
   1:L PR[91] R[100]mm/sec CNT100;
   1:  PR[91,1] = PR[90,1] + 10.331;
   1:  PR[91,2] = PR[90,2] + -11.581;
   1:L PR[91] R[100]mm/sec CNT100;
   1:  PR[91,1] = PR[90,1] + 11.288;
   1:  PR[91,2] = PR[90,2] + -12.826;
   1:L PR[91] R[100]mm/sec CNT100;
   1:  PR[91,1] = PR[90,1] + 12.770;
   1:  PR[91,2] = PR[90,2] + -14.307;
   1:L PR[91] R[100]mm/sec CNT100;
   1:  PR[91,1] = PR[90,1] + 14.003;
   1:  PR[91,2] = PR[90,2] + -15.250;
   1:L PR[91] R[100]mm/sec CNT100;
   1:  PR[91,1] = PR[90,1] + 15.771;
   1:  PR[91,2] = PR[90,2] + -16.487;
   1:L PR[91] R[100]mm/sec CNT100;
   1:  PR[91,1] = PR[90,1] + 17.719;
   1:  PR[91,2] = PR[90,2] + -17.395;
   1:L PR[91] R[100]mm/sec CNT100;
   1:  PR[91,1] = PR[90,1] + 19.143;
   1:  PR[91,2] = PR[90,2] + -17.982;
   1:L PR[91] R[100]mm/sec CNT100;
   1:  PR[91,1] = PR[90,1] + 21.194;
   1:  PR[91,2] = PR[90,2] + -18.531;
   1:L PR[91] R[100]mm/sec CNT100;
   1:  PR[91,1] = PR[90,1] + 22.698;
   1:  PR[91,2] = PR[90,2] + -18.727;
   1:L PR[91] R[100]mm/sec CNT100;
   1:  PR[91,1] = PR[90,1] + 24.867;
   1:  PR[91,2] = PR[90,2] + -18.915;
   1:L PR[91] R[100]mm/sec CNT100;
   1:  PR[91,1] = PR[90,1] + 27.032;
   1:  PR[91,2] = PR[90,2] + -18.725;
   1:L PR[91] R[100]mm/sec CNT100;
   1:  PR[91,1] = PR[90,1] + 28.522;
   1:  PR[91,2] = PR[90,2] + -18.526;
   1:L PR[91] R[100]mm/sec CNT100;
   1:  PR[91,1] = PR[90,1] + 30.554;
   1:  PR[91,2] = PR[90,2] + -17.981;
   1:L PR[91] R[100]mm/sec CNT100;
   1:  PR[91,1] = PR[90,1] + 32.611;
   1:  PR[91,2] = PR[90,2] + -17.022;
   1:L PR[91] R[100]mm/sec CNT100;
   1:  PR[91,1] = PR[90,1] + 33.986;
   1:  PR[91,2] = PR[90,2] + -16.449;
   1:L PR[91] R[100]mm/sec CNT100;
   1:  PR[91,1] = PR[90,1] + 35.754;
   1:  PR[91,2] = PR[90,2] + -15.211;
   1:L PR[91] R[100]mm/sec CNT100;
   1:  PR[91,1] = PR[90,1] + 36.919;
   1:  PR[91,2] = PR[90,2] + -14.315;
   1:L PR[91] R[100]mm/sec CNT100;
   1:  PR[91,1] = PR[90,1] + 38.447;
   1:  PR[91,2] = PR[90,2] + -12.788;
   1:L PR[91] R[100]mm/sec CNT100;
   1:  PR[91,1] = PR[90,1] + 39.330;
   1:  PR[91,2] = PR[90,2] + -11.634;
   1:L PR[91] R[100]mm/sec CNT100;
   1:  PR[91,1] = PR[90,1] + 40.603;
   1:  PR[91,2] = PR[90,2] + -9.815;
   1:L PR[91] R[100]mm/sec CNT100;
   1:  PR[91,1] = PR[90,1] + 41.538;
   1:  PR[91,2] = PR[90,2] + -7.810;
   1:L PR[91] R[100]mm/sec CNT100;
   1:  PR[91,1] = PR[90,1] + 42.091;
   1:  PR[91,2] = PR[90,2] + -6.473;
   1:L PR[91] R[100]mm/sec CNT100;
   1:  PR[91,1] = PR[90,1] + 42.643;
   1:  PR[91,2] = PR[90,2] + -4.410;
   1:L PR[91] R[100]mm/sec CNT100;
   1:  PR[91,1] = PR[90,1] + 42.843;
   1:  PR[91,2] = PR[90,2] + -2.130;
   1:L PR[91] R[100]mm/sec CNT100;
   1:  PR[91,1] = PR[90,1] + 43.009;
   1:  PR[91,2] = PR[90,2] + -0.700;
   1:L PR[91] R[100]mm/sec CNT100;
   1:  PR[91,1] = PR[90,1] + 42.838;
   1:  PR[91,2] = PR[90,2] + 1.265;
   1:L PR[91] R[100]mm/sec CNT100;
   1:  PR[91,1] = PR[90,1] + 42.833;
   1:  PR[91,2] = PR[90,2] + 1.549;
   1:L PR[91] R[100]mm/sec CNT100;
   1:  PR[91,1] = PR[90,1] + 42.655;
   1:  PR[91,2] = PR[90,2] + 2.909;
   1:L PR[91] R[100]mm/sec CNT100;
   1:  PR[91,1] = PR[90,1] + 42.091;
   1:  PR[91,2] = PR[90,2] + 5.015;
   1:L PR[91] R[100]mm/sec CNT100;
   1:  PR[91,1] = PR[90,1] + 41.538;
   1:  PR[91,2] = PR[90,2] + 6.352;
   1:L PR[91] R[100]mm/sec CNT100TB   .50sec,CALL END_PUD;
   1:  PR[92] = PR[91];
   1:  PR[92,3] = PR[92,3] + 20;
   1:J PR[92] 10% FINE;
   1:  PR[91,1] = PR[90,1] + 59.951;
   1:  PR[91,2] = PR[90,2] + -11.349;
   1:  PR[92] = PR[91];
   1:  PR[92,3] = PR[92,3] + 20;
   1:J PR[92] 10% FINE;
   1:L PR[91] R[100]mm/sec CNT100;
   1:  CALL LASER_DRAHT_START;
   1:  PR[91,1] = PR[90,1] + 60.519;
   1:  PR[91,2] = PR[90,2] + -12.161;
   1:L PR[91] R[100]mm/sec CNT100;
   1:  PR[91,1] = PR[90,1] + 63.218;
   1:  PR[91,2] = PR[90,2] + -14.844;
   1:L PR[91] R[100]mm/sec CNT100;
   1:  PR[91,1] = PR[90,1] + 64.125;
   1:  PR[91,2] = PR[90,2] + -15.479;
   1:L PR[91] R[100]mm/sec CNT100;
   1:  PR[91,1] = PR[90,1] + 66.314;
   1:  PR[91,2] = PR[90,2] + -16.842;
   1:L PR[91] R[100]mm/sec CNT100;
   1:  PR[91,1] = PR[90,1] + 67.427;
   1:  PR[91,2] = PR[90,2] + -17.362;
   1:L PR[91] R[100]mm/sec CNT100;
   1:  PR[91,1] = PR[90,1] + 69.676;
   1:  PR[91,2] = PR[90,2] + -18.138;
   1:L PR[91] R[100]mm/sec CNT100;
   1:  PR[91,1] = PR[90,1] + 70.966;
   1:  PR[91,2] = PR[90,2] + -18.484;
   1:L PR[91] R[100]mm/sec CNT100;
   1:  PR[91,1] = PR[90,1] + 72.384;
   1:  PR[91,2] = PR[90,2] + -18.608;
   1:L PR[91] R[100]mm/sec CNT100;
   1:  PR[91,1] = PR[90,1] + 74.676;
   1:  PR[91,2] = PR[90,2] + -18.854;
   1:L PR[91] R[100]mm/sec CNT100;
   1:  PR[91,1] = PR[90,1] + 76.141;
   1:  PR[91,2] = PR[90,2] + -18.727;
   1:L PR[91] R[100]mm/sec CNT100;
   1:  PR[91,1] = PR[90,1] + 78.252;
   1:  PR[91,2] = PR[90,2] + -18.479;
   1:L PR[91] R[100]mm/sec CNT100;
   1:  PR[91,1] = PR[90,1] + 79.774;
   1:  PR[91,2] = PR[90,2] + -18.072;
   1:L PR[91] R[100]mm/sec CNT100;
   1:  PR[91,1] = PR[90,1] + 81.632;
   1:  PR[91,2] = PR[90,2] + -17.415;
   1:L PR[91] R[100]mm/sec CNT100;
   1:  PR[91,1] = PR[90,1] + 83.135;
   1:  PR[91,2] = PR[90,2] + -16.715;
   1:L PR[91] R[100]mm/sec CNT100;
   1:  PR[91,1] = PR[90,1] + 84.695;
   1:  PR[91,2] = PR[90,2] + -15.728;
   1:L PR[91] R[100]mm/sec CNT100;
   1:  PR[91,1] = PR[90,1] + 86.116;
   1:  PR[91,2] = PR[90,2] + -14.733;
   1:L PR[91] R[100]mm/sec CNT100;
   1:  PR[91,1] = PR[90,1] + 88.647;
   1:  PR[91,2] = PR[90,2] + -12.196;
   1:L PR[91] R[100]mm/sec CNT100;
   1:  PR[91,1] = PR[90,1] + 89.674;
   1:  PR[91,2] = PR[90,2] + -10.730;
   1:L PR[91] R[100]mm/sec CNT100;
   1:  PR[91,1] = PR[90,1] + 90.590;
   1:  PR[91,2] = PR[90,2] + -9.268;
   1:L PR[91] R[100]mm/sec CNT100;
   1:  PR[91,1] = PR[90,1] + 91.361;
   1:  PR[91,2] = PR[90,2] + -7.614;
   1:L PR[91] R[100]mm/sec CNT100;
   1:  PR[91,1] = PR[90,1] + 91.912;
   1:  PR[91,2] = PR[90,2] + -6.032;
   1:L PR[91] R[100]mm/sec CNT100;
   1:  PR[91,1] = PR[90,1] + 92.385;
   1:  PR[91,2] = PR[90,2] + -4.268;
   1:L PR[91] R[100]mm/sec CNT100;
   1:  PR[91,1] = PR[90,1] + 92.552;
   1:  PR[91,2] = PR[90,2] + -2.358;
   1:L PR[91] R[100]mm/sec CNT100;
   1:  PR[91,1] = PR[90,1] + 92.735;
   1:  PR[91,2] = PR[90,2] + -0.706;
   1:L PR[91] R[100]mm/sec CNT100;
   1:  PR[91,1] = PR[90,1] + 92.571;
   1:  PR[91,2] = PR[90,2] + 1.163;
   1:L PR[91] R[100]mm/sec CNT100;
   1:  PR[91,1] = PR[90,1] + 92.391;
   1:  PR[91,2] = PR[90,2] + 2.786;
   1:L PR[91] R[100]mm/sec CNT100;
   1:  PR[91,1] = PR[90,1] + 91.912;
   1:  PR[91,2] = PR[90,2] + 4.572;
   1:L PR[91] R[100]mm/sec CNT100;
   1:  PR[91,1] = PR[90,1] + 91.361;
   1:  PR[91,2] = PR[90,2] + 6.155;
   1:L PR[91] R[100]mm/sec CNT100;
   1:  PR[91,1] = PR[90,1] + 90.591;
   1:  PR[91,2] = PR[90,2] + 7.807;
   1:L PR[91] R[100]mm/sec CNT100;
   1:  PR[91,1] = PR[90,1] + 89.675;
   1:  PR[91,2] = PR[90,2] + 9.270;
   1:L PR[91] R[100]mm/sec CNT100;
   1:  PR[91,1] = PR[90,1] + 88.649;
   1:  PR[91,2] = PR[90,2] + 10.735;
   1:L PR[91] R[100]mm/sec CNT100;
   1:  PR[91,1] = PR[90,1] + 86.119;
   1:  PR[91,2] = PR[90,2] + 13.272;
   1:L PR[91] R[100]mm/sec CNT100;
   1:  PR[91,1] = PR[90,1] + 84.698;
   1:  PR[91,2] = PR[90,2] + 14.267;
   1:L PR[91] R[100]mm/sec CNT100;
   1:  PR[91,1] = PR[90,1] + 83.138;
   1:  PR[91,2] = PR[90,2] + 15.254;
   1:L PR[91] R[100]mm/sec CNT100;
   1:  PR[91,1] = PR[90,1] + 81.637;
   1:  PR[91,2] = PR[90,2] + 15.955;
   1:L PR[91] R[100]mm/sec CNT100;
   1:  PR[91,1] = PR[90,1] + 79.779;
   1:  PR[91,2] = PR[90,2] + 16.611;
   1:L PR[91] R[100]mm/sec CNT100;
   1:  PR[91,1] = PR[90,1] + 78.286;
   1:  PR[91,2] = PR[90,2] + 17.012;
   1:L PR[91] R[100]mm/sec CNT100;
   1:  PR[91,1] = PR[90,1] + 76.640;
   1:  PR[91,2] = PR[90,2] + 17.156;
   1:L PR[91] R[100]mm/sec CNT100;
   1:  PR[91,1] = PR[90,1] + 74.632;
   1:  PR[91,2] = PR[90,2] + 17.395;
   1:L PR[91] R[100]mm/sec CNT100;
   1:  PR[91,1] = PR[90,1] + 73.168;
   1:  PR[91,2] = PR[90,2] + 17.267;
   1:L PR[91] R[100]mm/sec CNT100;
   1:  PR[91,1] = PR[90,1] + 70.991;
   1:  PR[91,2] = PR[90,2] + 17.031;
   1:L PR[91] R[100]mm/sec CNT100;
   1:  PR[91,1] = PR[90,1] + 69.680;
   1:  PR[91,2] = PR[90,2] + 16.681;
   1:L PR[91] R[100]mm/sec CNT100;
   1:  PR[91,1] = PR[90,1] + 67.431;
   1:  PR[91,2] = PR[90,2] + 15.904;
   1:L PR[91] R[100]mm/sec CNT100;
   1:  PR[91,1] = PR[90,1] + 66.317;
   1:  PR[91,2] = PR[90,2] + 15.385;
   1:L PR[91] R[100]mm/sec CNT100;
   1:  PR[91,1] = PR[90,1] + 64.127;
   1:  PR[91,2] = PR[90,2] + 14.021;
   1:L PR[91] R[100]mm/sec CNT100;
   1:  PR[91,1] = PR[90,1] + 63.220;
   1:  PR[91,2] = PR[90,2] + 13.387;
   1:L PR[91] R[100]mm/sec CNT100;
   1:  PR[91,1] = PR[90,1] + 60.520;
   1:  PR[91,2] = PR[90,2] + 10.704;
   1:L PR[91] R[100]mm/sec CNT100;
   1:  PR[91,1] = PR[90,1] + 59.952;
   1:  PR[91,2] = PR[90,2] + 9.892;
   1:L PR[91] R[100]mm/sec CNT100;
   1:  PR[91,1] = PR[90,1] + 58.438;
   1:  PR[91,2] = PR[90,2] + 7.499;
   1:L PR[91] R[100]mm/sec CNT100;
   1:  PR[91,1] = PR[90,1] + 58.062;
   1:  PR[91,2] = PR[90,2] + 6.693;
   1:L PR[91] R[100]mm/sec CNT100;
   1:  PR[91,1] = PR[90,1] + 57.080;
   1:  PR[91,2] = PR[90,2] + 3.898;
   1:L PR[91] R[100]mm/sec CNT100;
   1:  PR[91,1] = PR[90,1] + 56.872;
   1:  PR[91,2] = PR[90,2] + 3.124;
   1:L PR[91] R[100]mm/sec CNT100;
   1:  PR[91,1] = PR[90,1] + 56.794;
   1:  PR[91,2] = PR[90,2] + 2.226;
   1:L PR[91] R[100]mm/sec CNT100;
   1:  PR[91,1] = PR[90,1] + 56.457;
   1:  PR[91,2] = PR[90,2] + -0.755;
   1:L PR[91] R[100]mm/sec CNT100;
   1:  PR[91,1] = PR[90,1] + 56.526;
   1:  PR[91,2] = PR[90,2] + -1.538;
   1:L PR[91] R[100]mm/sec CNT100;
   1:  PR[91,1] = PR[90,1] + 56.866;
   1:  PR[91,2] = PR[90,2] + -4.558;
   1:L PR[91] R[100]mm/sec CNT100;
   1:  PR[91,1] = PR[90,1] + 57.079;
   1:  PR[91,2] = PR[90,2] + -5.357;
   1:L PR[91] R[100]mm/sec CNT100;
   1:  PR[91,1] = PR[90,1] + 58.062;
   1:  PR[91,2] = PR[90,2] + -8.151;
   1:L PR[91] R[100]mm/sec CNT100;
   1:  PR[91,1] = PR[90,1] + 58.438;
   1:  PR[91,2] = PR[90,2] + -8.957;
   1:L PR[91] R[100]mm/sec CNT100;
   1:  PR[91,1] = PR[90,1] + 59.951;
   1:  PR[91,2] = PR[90,2] + -11.349;
   1:L PR[91] R[100]mm/sec CNT100TB   .50sec,CALL END_PUD;
   1:  PR[92] = PR[91];
   1:  PR[92,3] = PR[92,3] + 20;
   1:J PR[92] 10% FINE;
   1:  PR[91,1] = PR[90,1] + -38.808;
   1:  PR[91,2] = PR[90,2] + -12.219;
   1:  PR[92] = PR[91];
   1:  PR[92,3] = PR[92,3] + 20;
   1:J PR[92] 10% FINE;
   1:L PR[91] R[100]mm/sec CNT100;
   1:  CALL LASER_DRAHT_START;
   1:  PR[91,1] = PR[90,1] + -36.340;
   1:  PR[91,2] = PR[90,2] + -14.691;
   1:L PR[91] R[100]mm/sec CNT100;
   1:  PR[91,1] = PR[90,1] + -34.645;
   1:  PR[91,2] = PR[90,2] + -15.878;
   1:L PR[91] R[100]mm/sec CNT100;
   1:  PR[91,1] = PR[90,1] + -33.468;
   1:  PR[91,2] = PR[90,2] + -16.622;
   1:L PR[91] R[100]mm/sec CNT100;
   1:  PR[91,1] = PR[90,1] + -31.623;
   1:  PR[91,2] = PR[90,2] + -17.483;
   1:L PR[91] R[100]mm/sec CNT100;
   1:  PR[91,1] = PR[90,1] + -30.253;
   1:  PR[91,2] = PR[90,2] + -17.966;
   1:L PR[91] R[100]mm/sec CNT100;
   1:  PR[91,1] = PR[90,1] + -28.354;
   1:  PR[91,2] = PR[90,2] + -18.475;
   1:L PR[91] R[100]mm/sec CNT100;
   1:  PR[91,1] = PR[90,1] + -26.288;
   1:  PR[91,2] = PR[90,2] + -18.656;
   1:L PR[91] R[100]mm/sec CNT100;
   1:  PR[91,1] = PR[90,1] + -24.821;
   1:  PR[91,2] = PR[90,2] + -18.828;
   1:L PR[91] R[100]mm/sec CNT100;
   1:  PR[91,1] = PR[90,1] + -22.881;
   1:  PR[91,2] = PR[90,2] + -18.658;
   1:L PR[91] R[100]mm/sec CNT100;
   1:  PR[91,1] = PR[90,1] + -21.338;
   1:  PR[91,2] = PR[90,2] + -18.489;
   1:L PR[91] R[100]mm/sec CNT100;
   1:  PR[91,1] = PR[90,1] + -19.504;
   1:  PR[91,2] = PR[90,2] + -17.997;
   1:L PR[91] R[100]mm/sec CNT100;
   1:  PR[91,1] = PR[90,1] + -17.962;
   1:  PR[91,2] = PR[90,2] + -17.463;
   1:L PR[91] R[100]mm/sec CNT100;
   1:  PR[91,1] = PR[90,1] + -16.287;
   1:  PR[91,2] = PR[90,2] + -16.682;
   1:L PR[91] R[100]mm/sec CNT100;
   1:  PR[91,1] = PR[90,1] + -14.835;
   1:  PR[91,2] = PR[90,2] + -15.775;
   1:L PR[91] R[100]mm/sec CNT100;
   1:  PR[91,1] = PR[90,1] + -13.364;
   1:  PR[91,2] = PR[90,2] + -14.745;
   1:L PR[91] R[100]mm/sec CNT100;
   1:  PR[91,1] = PR[90,1] + -10.822;
   1:  PR[91,2] = PR[90,2] + -12.210;
   1:L PR[91] R[100]mm/sec CNT100;
   1:  PR[91,1] = PR[90,1] + -9.816;
   1:  PR[91,2] = PR[90,2] + -10.772;
   1:L PR[91] R[100]mm/sec CNT100;
   1:  PR[91,1] = PR[90,1] + -8.852;
   1:  PR[91,2] = PR[90,2] + -9.245;
   1:L PR[91] R[100]mm/sec CNT100;
   1:  PR[91,1] = PR[90,1] + -8.125;
   1:  PR[91,2] = PR[90,2] + -7.685;
   1:L PR[91] R[100]mm/sec CNT100;
   1:  PR[91,1] = PR[90,1] + -7.512;
   1:  PR[91,2] = PR[90,2] + -5.937;
   1:L PR[91] R[100]mm/sec CNT100;
   1:  PR[91,1] = PR[90,1] + -7.079;
   1:  PR[91,2] = PR[90,2] + -4.322;
   1:L PR[91] R[100]mm/sec CNT100;
   1:  PR[91,1] = PR[90,1] + -6.926;
   1:  PR[91,2] = PR[90,2] + -2.566;
   1:L PR[91] R[100]mm/sec CNT100;
   1:  PR[91,1] = PR[90,1] + -6.733;
   1:  PR[91,2] = PR[90,2] + -0.713;
   1:L PR[91] R[100]mm/sec CNT100;
   1:  PR[91,1] = PR[90,1] + -6.894;
   1:  PR[91,2] = PR[90,2] + 1.132;
   1:L PR[91] R[100]mm/sec CNT100;
   1:  PR[91,1] = PR[90,1] + -6.886;
   1:  PR[91,2] = PR[90,2] + 1.192;
   1:L PR[91] R[100]mm/sec CNT100;
   1:  PR[91,1] = PR[90,1] + -7.073;
   1:  PR[91,2] = PR[90,2] + 2.838;
   1:L PR[91] R[100]mm/sec CNT100;
   1:  PR[91,1] = PR[90,1] + -7.512;
   1:  PR[91,2] = PR[90,2] + 4.478;
   1:L PR[91] R[100]mm/sec CNT100;
   1:  PR[91,1] = PR[90,1] + -8.125;
   1:  PR[91,2] = PR[90,2] + 6.226;
   1:L PR[91] R[100]mm/sec CNT100;
   1:  PR[91,1] = PR[90,1] + -8.852;
   1:  PR[91,2] = PR[90,2] + 7.785;
   1:L PR[91] R[100]mm/sec CNT100;
   1:  PR[91,1] = PR[90,1] + -9.816;
   1:  PR[91,2] = PR[90,2] + 9.313;
   1:L PR[91] R[100]mm/sec CNT100;
   1:  PR[91,1] = PR[90,1] + -10.822;
   1:  PR[91,2] = PR[90,2] + 10.750;
   1:L PR[91] R[100]mm/sec CNT100;
   1:  PR[91,1] = PR[90,1] + -13.364;
   1:  PR[91,2] = PR[90,2] + 13.285;
   1:L PR[91] R[100]mm/sec CNT100;
   1:  PR[91,1] = PR[90,1] + -14.834;
   1:  PR[91,2] = PR[90,2] + 14.315;
   1:L PR[91] R[100]mm/sec CNT100;
   1:  PR[91,1] = PR[90,1] + -16.286;
   1:  PR[91,2] = PR[90,2] + 15.223;
   1:L PR[91] R[100]mm/sec CNT100;
   1:  PR[91,1] = PR[90,1] + -17.961;
   1:  PR[91,2] = PR[90,2] + 16.004;
   1:L PR[91] R[100]mm/sec CNT100;
   1:  PR[91,1] = PR[90,1] + -19.504;
   1:  PR[91,2] = PR[90,2] + 16.538;
   1:L PR[91] R[100]mm/sec CNT100;
   1:  PR[91,1] = PR[90,1] + -21.316;
   1:  PR[91,2] = PR[90,2] + 17.024;
   1:L PR[91] R[100]mm/sec CNT100;
   1:  PR[91,1] = PR[90,1] + -23.278;
   1:  PR[91,2] = PR[90,2] + 17.196;
   1:L PR[91] R[100]mm/sec CNT100;
   1:  PR[91,1] = PR[90,1] + -24.870;
   1:  PR[91,2] = PR[90,2] + 17.370;
   1:L PR[91] R[100]mm/sec CNT100;
   1:  PR[91,1] = PR[90,1] + -26.812;
   1:  PR[91,2] = PR[90,2] + 17.200;
   1:L PR[91] R[100]mm/sec CNT100;
   1:  PR[91,1] = PR[90,1] + -28.325;
   1:  PR[91,2] = PR[90,2] + 17.024;
   1:L PR[91] R[100]mm/sec CNT100;
   1:  PR[91,1] = PR[90,1] + -30.252;
   1:  PR[91,2] = PR[90,2] + 16.507;
   1:L PR[91] R[100]mm/sec CNT100;
   1:  PR[91,1] = PR[90,1] + -31.622;
   1:  PR[91,2] = PR[90,2] + 16.024;
   1:L PR[91] R[100]mm/sec CNT100;
   1:  PR[91,1] = PR[90,1] + -33.467;
   1:  PR[91,2] = PR[90,2] + 15.164;
   1:L PR[91] R[100]mm/sec CNT100;
   1:  PR[91,1] = PR[90,1] + -34.645;
   1:  PR[91,2] = PR[90,2] + 14.420;
   1:L PR[91] R[100]mm/sec CNT100;
   1:  PR[91,1] = PR[90,1] + -36.339;
   1:  PR[91,2] = PR[90,2] + 13.233;
   1:L PR[91] R[100]mm/sec CNT100;
   1:  PR[91,1] = PR[90,1] + -38.807;
   1:  PR[91,2] = PR[90,2] + 10.760;
   1:L PR[91] R[100]mm/sec CNT100;
   1:  PR[91,1] = PR[90,1] + -40.008;
   1:  PR[91,2] = PR[90,2] + 9.044;
   1:L PR[91] R[100]mm/sec CNT100;
   1:  PR[91,1] = PR[90,1] + -40.716;
   1:  PR[91,2] = PR[90,2] + 7.915;
   1:L PR[91] R[100]mm/sec CNT100;
   1:  PR[91,1] = PR[90,1] + -41.611;
   1:  PR[91,2] = PR[90,2] + 5.995;
   1:L PR[91] R[100]mm/sec CNT100;
   1:  PR[91,1] = PR[90,1] + -42.041;
   1:  PR[91,2] = PR[90,2] + 4.761;
   1:L PR[91] R[100]mm/sec CNT100;
   1:  PR[91,1] = PR[90,1] + -42.585;
   1:  PR[91,2] = PR[90,2] + 2.729;
   1:L PR[91] R[100]mm/sec CNT100;
   1:  PR[91,1] = PR[90,1] + -42.777;
   1:  PR[91,2] = PR[90,2] + 0.537;
   1:L PR[91] R[100]mm/sec CNT100;
   1:  PR[91,1] = PR[90,1] + -42.922;
   1:  PR[91,2] = PR[90,2] + -0.754;
   1:L PR[91] R[100]mm/sec CNT100;
   1:  PR[91,1] = PR[90,1] + -42.736;
   1:  PR[91,2] = PR[90,2] + -2.878;
   1:L PR[91] R[100]mm/sec CNT100;
   1:  PR[91,1] = PR[90,1] + -42.592;
   1:  PR[91,2] = PR[90,2] + -4.163;
   1:L PR[91] R[100]mm/sec CNT100;
   1:  PR[91,1] = PR[90,1] + -42.041;
   1:  PR[91,2] = PR[90,2] + -6.219;
   1:L PR[91] R[100]mm/sec CNT100;
   1:  PR[91,1] = PR[90,1] + -41.611;
   1:  PR[91,2] = PR[90,2] + -7.453;
   1:L PR[91] R[100]mm/sec CNT100;
   1:  PR[91,1] = PR[90,1] + -40.716;
   1:  PR[91,2] = PR[90,2] + -9.373;
   1:L PR[91] R[100]mm/sec CNT100;
   1:  PR[91,1] = PR[90,1] + -40.009;
   1:  PR[91,2] = PR[90,2] + -10.502;
   1:L PR[91] R[100]mm/sec CNT100;
   1:  PR[91,1] = PR[90,1] + -38.808;
   1:  PR[91,2] = PR[90,2] + -12.219;
   1:L PR[91] R[100]mm/sec CNT100TB   .50sec,CALL END_PUD;
   1:  PR[92] = PR[91];
   1:  PR[92,3] = PR[92,3] + 20;
   1:J PR[92] 10% FINE;
   1:  PR[91,1] = PR[90,1] + -92.519;
   1:  PR[91,2] = PR[90,2] + -4.101;
   1:  PR[92] = PR[91];
   1:  PR[92,3] = PR[92,3] + 20;
   1:J PR[92] 10% FINE;
   1:L PR[91] R[100]mm/sec CNT100;
   1:  CALL LASER_DRAHT_START;
   1:  PR[91,1] = PR[90,1] + -92.006;
   1:  PR[91,2] = PR[90,2] + -6.016;
   1:L PR[91] R[100]mm/sec CNT100;
   1:  PR[91,1] = PR[90,1] + -91.574;
   1:  PR[91,2] = PR[90,2] + -7.348;
   1:L PR[91] R[100]mm/sec CNT100;
   1:  PR[91,1] = PR[90,1] + -90.745;
   1:  PR[91,2] = PR[90,2] + -9.125;
   1:L PR[91] R[100]mm/sec CNT100;
   1:  PR[91,1] = PR[90,1] + -90.030;
   1:  PR[91,2] = PR[90,2] + -10.365;
   1:L PR[91] R[100]mm/sec CNT100;
   1:  PR[91,1] = PR[90,1] + -88.918;
   1:  PR[91,2] = PR[90,2] + -11.953;
   1:L PR[91] R[100]mm/sec CNT100;
   1:  PR[91,1] = PR[90,1] + -87.928;
   1:  PR[91,2] = PR[90,2] + -13.056;
   1:L PR[91] R[100]mm/sec CNT100;
   1:  PR[91,1] = PR[90,1] + -86.592;
   1:  PR[91,2] = PR[90,2] + -14.391;
   1:L PR[91] R[100]mm/sec CNT100;
   1:  PR[91,1] = PR[90,1] + -85.338;
   1:  PR[91,2] = PR[90,2] + -15.306;
   1:L PR[91] R[100]mm/sec CNT100;
   1:  PR[91,1] = PR[90,1] + -83.816;
   1:  PR[91,2] = PR[90,2] + -16.371;
   1:L PR[91] R[100]mm/sec CNT100;
   1:  PR[91,1] = PR[90,1] + -82.132;
   1:  PR[91,2] = PR[90,2] + -17.155;
   1:L PR[91] R[100]mm/sec CNT100;
   1:  PR[91,1] = PR[90,1] + -80.695;
   1:  PR[91,2] = PR[90,2] + -17.799;
   1:L PR[91] R[100]mm/sec CNT100;
   1:  PR[91,1] = PR[90,1] + -78.979;
   1:  PR[91,2] = PR[90,2] + -18.258;
   1:L PR[91] R[100]mm/sec CNT100;
   1:  PR[91,1] = PR[90,1] + -77.345;
   1:  PR[91,2] = PR[90,2] + -18.609;
   1:L PR[91] R[100]mm/sec CNT100;
   1:  PR[91,1] = PR[90,1] + -75.652;
   1:  PR[91,2] = PR[90,2] + -18.757;
   1:L PR[91] R[100]mm/sec CNT100;
   1:  PR[91,1] = PR[90,1] + -73.868;
   1:  PR[91,2] = PR[90,2] + -18.761;
   1:L PR[91] R[100]mm/sec CNT100;
   1:  PR[91,1] = PR[90,1] + -72.260;
   1:  PR[91,2] = PR[90,2] + -18.620;
   1:L PR[91] R[100]mm/sec CNT100;
   1:  PR[91,1] = PR[90,1] + -70.389;
   1:  PR[91,2] = PR[90,2] + -18.227;
   1:L PR[91] R[100]mm/sec CNT100;
   1:  PR[91,1] = PR[90,1] + -68.939;
   1:  PR[91,2] = PR[90,2] + -17.838;
   1:L PR[91] R[100]mm/sec CNT100;
   1:  PR[91,1] = PR[90,1] + -67.513;
   1:  PR[91,2] = PR[90,2] + -17.172;
   1:L PR[91] R[100]mm/sec CNT100;
   1:  PR[91,1] = PR[90,1] + -65.729;
   1:  PR[91,2] = PR[90,2] + -16.385;
   1:L PR[91] R[100]mm/sec CNT100;
   1:  PR[91,1] = PR[90,1] + -64.561;
   1:  PR[91,2] = PR[90,2] + -15.568;
   1:L PR[91] R[100]mm/sec CNT100;
   1:  PR[91,1] = PR[90,1] + -62.869;
   1:  PR[91,2] = PR[90,2] + -14.346;
   1:L PR[91] R[100]mm/sec CNT100;
   1:  PR[91,1] = PR[90,1] + -61.932;
   1:  PR[91,2] = PR[90,2] + -13.409;
   1:L PR[91] R[100]mm/sec CNT100;
   1:  PR[91,1] = PR[90,1] + -60.445;
   1:  PR[91,2] = PR[90,2] + -11.763;
   1:L PR[91] R[100]mm/sec CNT100;
   1:  PR[91,1] = PR[90,1] + -59.730;
   1:  PR[91,2] = PR[90,2] + -10.742;
   1:L PR[91] R[100]mm/sec CNT100;
   1:  PR[91,1] = PR[90,1] + -58.562;
   1:  PR[91,2] = PR[90,2] + -8.726;
   1:L PR[91] R[100]mm/sec CNT100;
   1:  PR[91,1] = PR[90,1] + -58.067;
   1:  PR[91,2] = PR[90,2] + -7.664;
   1:L PR[91] R[100]mm/sec CNT100;
   1:  PR[91,1] = PR[90,1] + -57.321;
   1:  PR[91,2] = PR[90,2] + -5.374;
   1:L PR[91] R[100]mm/sec CNT100;
   1:  PR[91,1] = PR[90,1] + -57.033;
   1:  PR[91,2] = PR[90,2] + -4.298;
   1:L PR[91] R[100]mm/sec CNT100;
   1:  PR[91,1] = PR[90,1] + -56.714;
   1:  PR[91,2] = PR[90,2] + -0.727;
   1:L PR[91] R[100]mm/sec CNT100;
   1:  PR[91,1] = PR[90,1] + -56.791;
   1:  PR[91,2] = PR[90,2] + 0.155;
   1:L PR[91] R[100]mm/sec CNT100;
   1:  PR[91,1] = PR[90,1] + -57.078;
   1:  PR[91,2] = PR[90,2] + 2.868;
   1:L PR[91] R[100]mm/sec CNT100;
   1:  PR[91,1] = PR[90,1] + -57.309;
   1:  PR[91,2] = PR[90,2] + 3.730;
   1:L PR[91] R[100]mm/sec CNT100;
   1:  PR[91,1] = PR[90,1] + -58.141;
   1:  PR[91,2] = PR[90,2] + 6.288;
   1:L PR[91] R[100]mm/sec CNT100;
   1:  PR[91,1] = PR[90,1] + -58.538;
   1:  PR[91,2] = PR[90,2] + 7.140;
   1:L PR[91] R[100]mm/sec CNT100;
   1:  PR[91,1] = PR[90,1] + -59.842;
   1:  PR[91,2] = PR[90,2] + 9.392;
   1:L PR[91] R[100]mm/sec CNT100;
   1:  PR[91,1] = PR[90,1] + -60.428;
   1:  PR[91,2] = PR[90,2] + 10.228;
   1:L PR[91] R[100]mm/sec CNT100;
   1:  PR[91,1] = PR[90,1] + -62.089;
   1:  PR[91,2] = PR[90,2] + 12.068;
   1:L PR[91] R[100]mm/sec CNT100;
   1:  PR[91,1] = PR[90,1] + -62.874;
   1:  PR[91,2] = PR[90,2] + 12.853;
   1:L PR[91] R[100]mm/sec CNT100;
   1:  PR[91,1] = PR[90,1] + -64.766;
   1:  PR[91,2] = PR[90,2] + 14.221;
   1:L PR[91] R[100]mm/sec CNT100;
   1:  PR[91,1] = PR[90,1] + -65.781;
   1:  PR[91,2] = PR[90,2] + 14.932;
   1:L PR[91] R[100]mm/sec CNT100;
   1:  PR[91,1] = PR[90,1] + -66.898;
   1:  PR[91,2] = PR[90,2] + 15.452;
   1:L PR[91] R[100]mm/sec CNT100;
   1:  PR[91,1] = PR[90,1] + -68.993;
   1:  PR[91,2] = PR[90,2] + 16.380;
   1:L PR[91] R[100]mm/sec CNT100;
   1:  PR[91,1] = PR[90,1] + -70.275;
   1:  PR[91,2] = PR[90,2] + 16.723;
   1:L PR[91] R[100]mm/sec CNT100;
   1:  PR[91,1] = PR[90,1] + -72.370;
   1:  PR[91,2] = PR[90,2] + 17.164;
   1:L PR[91] R[100]mm/sec CNT100;
   1:  PR[91,1] = PR[90,1] + -73.793;
   1:  PR[91,2] = PR[90,2] + 17.288;
   1:L PR[91] R[100]mm/sec CNT100;
   1:  PR[91,1] = PR[90,1] + -75.793;
   1:  PR[91,2] = PR[90,2] + 17.285;
   1:L PR[91] R[100]mm/sec CNT100;
   1:  PR[91,1] = PR[90,1] + -77.309;
   1:  PR[91,2] = PR[90,2] + 17.152;
   1:L PR[91] R[100]mm/sec CNT100;
   1:  PR[91,1] = PR[90,1] + -79.143;
   1:  PR[91,2] = PR[90,2] + 16.759;
   1:L PR[91] R[100]mm/sec CNT100;
   1:  PR[91,1] = PR[90,1] + -80.680;
   1:  PR[91,2] = PR[90,2] + 16.347;
   1:L PR[91] R[100]mm/sec CNT100;
   1:  PR[91,1] = PR[90,1] + -82.179;
   1:  PR[91,2] = PR[90,2] + 15.648;
   1:L PR[91] R[100]mm/sec CNT100;
   1:  PR[91,1] = PR[90,1] + -83.858;
   1:  PR[91,2] = PR[90,2] + 14.895;
   1:L PR[91] R[100]mm/sec CNT100;
   1:  PR[91,1] = PR[90,1] + -85.235;
   1:  PR[91,2] = PR[90,2] + 13.931;
   1:L PR[91] R[100]mm/sec CNT100;
   1:  PR[91,1] = PR[90,1] + -86.643;
   1:  PR[91,2] = PR[90,2] + 12.905;
   1:L PR[91] R[100]mm/sec CNT100;
   1:  PR[91,1] = PR[90,1] + -87.869;
   1:  PR[91,2] = PR[90,2] + 11.679;
   1:L PR[91] R[100]mm/sec CNT100;
   1:  PR[91,1] = PR[90,1] + -88.981;
   1:  PR[91,2] = PR[90,2] + 10.441;
   1:L PR[91] R[100]mm/sec CNT100;
   1:  PR[91,1] = PR[90,1] + -90.006;
   1:  PR[91,2] = PR[90,2] + 8.977;
   1:L PR[91] R[100]mm/sec CNT100;
   1:  PR[91,1] = PR[90,1] + -90.810;
   1:  PR[91,2] = PR[90,2] + 7.583;
   1:L PR[91] R[100]mm/sec CNT100;
   1:  PR[91,1] = PR[90,1] + -91.576;
   1:  PR[91,2] = PR[90,2] + 5.941;
   1:L PR[91] R[100]mm/sec CNT100;
   1:  PR[91,1] = PR[90,1] + -92.061;
   1:  PR[91,2] = PR[90,2] + 4.443;
   1:L PR[91] R[100]mm/sec CNT100;
   1:  PR[91,1] = PR[90,1] + -92.532;
   1:  PR[91,2] = PR[90,2] + 2.686;
   1:L PR[91] R[100]mm/sec CNT100;
   1:  PR[91,1] = PR[90,1] + -92.696;
   1:  PR[91,2] = PR[90,2] + 0.810;
   1:L PR[91] R[100]mm/sec CNT100;
   1:  PR[91,1] = PR[90,1] + -92.859;
   1:  PR[91,2] = PR[90,2] + -0.747;
   1:L PR[91] R[100]mm/sec CNT100;
   1:  PR[91,1] = PR[90,1] + -92.710;
   1:  PR[91,2] = PR[90,2] + -2.445;
   1:L PR[91] R[100]mm/sec CNT100;
   1:  PR[91,1] = PR[90,1] + -92.679;
   1:  PR[91,2] = PR[90,2] + -2.570;
   1:L PR[91] R[100]mm/sec CNT100;
   1:  PR[91,1] = PR[90,1] + -92.519;
   1:  PR[91,2] = PR[90,2] + -4.101;
   1:L PR[91] R[100]mm/sec CNT100TB   .50sec,CALL END_PUD;
   1:  PR[92] = PR[91];
   1:  PR[92,3] = PR[92,3] + 20;
   1:J PR[92] 10% FINE;
   1:  PR[91] = PR[90];
   1:  PR[91,1] = PR[90,1] + 19.260;
   1:  PR[91,2] = PR[90,2] + -18.084;
   1:  PR[91,3] = PR[90,3] + 14.495;
   1:  PR[92] = PR[91];
   1:  PR[92,3] = PR[92,3] + 20;
   1:J PR[92] 10% FINE;
   1:L PR[91] R[100]mm/sec CNT100;
   1:  CALL LASER_DRAHT_START;
   1:  PR[91,1] = PR[90,1] + 21.006;
   1:  PR[91,2] = PR[90,2] + -18.551;
   1:L PR[91] R[100]mm/sec CNT100;
   1:  PR[91,1] = PR[90,1] + 22.989;
   1:  PR[91,2] = PR[90,2] + -18.809;
   1:L PR[91] R[100]mm/sec CNT100;
   1:  PR[91,1] = PR[90,1] + 24.847;
   1:  PR[91,2] = PR[90,2] + -18.971;
   1:L PR[91] R[100]mm/sec CNT100;
   1:  PR[91,1] = PR[90,1] + 26.702;
   1:  PR[91,2] = PR[90,2] + -18.808;
   1:L PR[91] R[100]mm/sec CNT100;
   1:  PR[91,1] = PR[90,1] + 28.668;
   1:  PR[91,2] = PR[90,2] + -18.545;
   1:L PR[91] R[100]mm/sec CNT100;
   1:  PR[91,1] = PR[90,1] + 30.401;
   1:  PR[91,2] = PR[90,2] + -18.081;
   1:L PR[91] R[100]mm/sec CNT100;
   1:  PR[91,1] = PR[90,1] + 32.178;
   1:  PR[91,2] = PR[90,2] + -17.251;
   1:L PR[91] R[100]mm/sec CNT100;
   1:  PR[91,1] = PR[90,1] + 33.994;
   1:  PR[91,2] = PR[90,2] + -16.495;
   1:L PR[91] R[100]mm/sec CNT100;
   1:  PR[91,1] = PR[90,1] + 35.511;
   1:  PR[91,2] = PR[90,2] + -15.433;
   1:L PR[91] R[100]mm/sec CNT100;
   1:  PR[91,1] = PR[90,1] + 37.049;
   1:  PR[91,2] = PR[90,2] + -14.250;
   1:L PR[91] R[100]mm/sec CNT100;
   1:  PR[91,1] = PR[90,1] + 38.362;
   1:  PR[91,2] = PR[90,2] + -12.937;
   1:L PR[91] R[100]mm/sec CNT100;
   1:  PR[91,1] = PR[90,1] + 39.529;
   1:  PR[91,2] = PR[90,2] + -11.413;
   1:L PR[91] R[100]mm/sec CNT100;
   1:  PR[91,1] = PR[90,1] + 40.629;
   1:  PR[91,2] = PR[90,2] + -9.841;
   1:L PR[91] R[100]mm/sec CNT100;
   1:  PR[91,1] = PR[90,1] + 41.437;
   1:  PR[91,2] = PR[90,2] + -8.109;
   1:L PR[91] R[100]mm/sec CNT100;
   1:  PR[91,1] = PR[90,1] + 42.167;
   1:  PR[91,2] = PR[90,2] + -6.343;
   1:L PR[91] R[100]mm/sec CNT100;
   1:  PR[91,1] = PR[90,1] + 42.642;
   1:  PR[91,2] = PR[90,2] + -4.570;
   1:L PR[91] R[100]mm/sec CNT100;
   1:  PR[91,1] = PR[90,1] + 42.815;
   1:  PR[91,2] = PR[90,2] + -2.589;
   1:L PR[91] R[100]mm/sec CNT100;
   1:  PR[91,1] = PR[90,1] + 43.035;
   1:  PR[91,2] = PR[90,2] + -0.700;
   1:L PR[91] R[100]mm/sec CNT100;
   1:  PR[91,1] = PR[90,1] + 42.898;
   1:  PR[91,2] = PR[90,2] + 0.873;
   1:L PR[91] R[100]mm/sec CNT100;
   1:  PR[91,1] = PR[90,1] + 42.892;
   1:  PR[91,2] = PR[90,2] + 1.251;
   1:L PR[91] R[100]mm/sec CNT100;
   1:  PR[91,1] = PR[90,1] + 42.653;
   1:  PR[91,2] = PR[90,2] + 3.069;
   1:L PR[91] R[100]mm/sec CNT100;
   1:  PR[91,1] = PR[90,1] + 42.167;
   1:  PR[91,2] = PR[90,2] + 4.885;
   1:L PR[91] R[100]mm/sec CNT100;
   1:  PR[91,1] = PR[90,1] + 41.437;
   1:  PR[91,2] = PR[90,2] + 6.651;
   1:L PR[91] R[100]mm/sec CNT100;
   1:  PR[91,1] = PR[90,1] + 40.628;
   1:  PR[91,2] = PR[90,2] + 8.384;
   1:L PR[91] R[100]mm/sec CNT100;
   1:  PR[91,1] = PR[90,1] + 39.527;
   1:  PR[91,2] = PR[90,2] + 9.957;
   1:L PR[91] R[100]mm/sec CNT100;
   1:  PR[91,1] = PR[90,1] + 38.361;
   1:  PR[91,2] = PR[90,2] + 11.480;
   1:L PR[91] R[100]mm/sec CNT100;
   1:  PR[91,1] = PR[90,1] + 37.046;
   1:  PR[91,2] = PR[90,2] + 12.794;
   1:L PR[91] R[100]mm/sec CNT100;
   1:  PR[91,1] = PR[90,1] + 35.508;
   1:  PR[91,2] = PR[90,2] + 13.977;
   1:L PR[91] R[100]mm/sec CNT100;
   1:  PR[91,1] = PR[90,1] + 33.955;
   1:  PR[91,2] = PR[90,2] + 15.063;
   1:L PR[91] R[100]mm/sec CNT100;
   1:  PR[91,1] = PR[90,1] + 32.240;
   1:  PR[91,2] = PR[90,2] + 15.862;
   1:L PR[91] R[100]mm/sec CNT100;
   1:  PR[91,1] = PR[90,1] + 30.436;
   1:  PR[91,2] = PR[90,2] + 16.613;
   1:L PR[91] R[100]mm/sec CNT100;
   1:  PR[91,1] = PR[90,1] + 28.660;
   1:  PR[91,2] = PR[90,2] + 17.088;
   1:L PR[91] R[100]mm/sec CNT100;
   1:  PR[91,1] = PR[90,1] + 26.694;
   1:  PR[91,2] = PR[90,2] + 17.351;
   1:L PR[91] R[100]mm/sec CNT100;
   1:  PR[91,1] = PR[90,1] + 24.840;
   1:  PR[91,2] = PR[90,2] + 17.512;
   1:L PR[91] R[100]mm/sec CNT100;
   1:  PR[91,1] = PR[90,1] + 22.982;
   1:  PR[91,2] = PR[90,2] + 17.349;
   1:L PR[91] R[100]mm/sec CNT100;
   1:  PR[91,1] = PR[90,1] + 20.999;
   1:  PR[91,2] = PR[90,2] + 17.091;
   1:L PR[91] R[100]mm/sec CNT100;
   1:  PR[91,1] = PR[90,1] + 19.298;
   1:  PR[91,2] = PR[90,2] + 16.635;
   1:L PR[91] R[100]mm/sec CNT100;
   1:  PR[91,1] = PR[90,1] + 17.545;
   1:  PR[91,2] = PR[90,2] + 15.817;
   1:L PR[91] R[100]mm/sec CNT100;
   1:  PR[91,1] = PR[90,1] + 15.681;
   1:  PR[91,2] = PR[90,2] + 15.049;
   1:L PR[91] R[100]mm/sec CNT100;
   1:  PR[91,1] = PR[90,1] + 14.213;
   1:  PR[91,2] = PR[90,2] + 14.021;
   1:L PR[91] R[100]mm/sec CNT100;
   1:  PR[91,1] = PR[90,1] + 12.588;
   1:  PR[91,2] = PR[90,2] + 12.778;
   1:L PR[91] R[100]mm/sec CNT100;
   1:  PR[91,1] = PR[90,1] + 11.334;
   1:  PR[91,2] = PR[90,2] + 11.524;
   1:L PR[91] R[100]mm/sec CNT100;
   1:  PR[91,1] = PR[90,1] + 10.073;
   1:  PR[91,2] = PR[90,2] + 9.883;
   1:L PR[91] R[100]mm/sec CNT100;
   1:  PR[91,1] = PR[90,1] + 9.032;
   1:  PR[91,2] = PR[90,2] + 8.397;
   1:L PR[91] R[100]mm/sec CNT100;
   1:  PR[91,1] = PR[90,1] + 8.267;
   1:  PR[91,2] = PR[90,2] + 6.756;
   1:L PR[91] R[100]mm/sec CNT100;
   1:  PR[91,1] = PR[90,1] + 7.471;
   1:  PR[91,2] = PR[90,2] + 4.837;
   1:L PR[91] R[100]mm/sec CNT100;
   1:  PR[91,1] = PR[90,1] + 7.026;
   1:  PR[91,2] = PR[90,2] + 3.176;
   1:L PR[91] R[100]mm/sec CNT100;
   1:  PR[91,1] = PR[90,1] + 6.861;
   1:  PR[91,2] = PR[90,2] + 1.294;
   1:L PR[91] R[100]mm/sec CNT100;
   1:  PR[91,1] = PR[90,1] + 6.592;
   1:  PR[91,2] = PR[90,2] + -0.772;
   1:L PR[91] R[100]mm/sec CNT100;
   1:  PR[91,1] = PR[90,1] + 6.753;
   1:  PR[91,2] = PR[90,2] + -2.611;
   1:L PR[91] R[100]mm/sec CNT100;
   1:  PR[91,1] = PR[90,1] + 7.014;
   1:  PR[91,2] = PR[90,2] + -4.592;
   1:L PR[91] R[100]mm/sec CNT100;
   1:  PR[91,1] = PR[90,1] + 7.471;
   1:  PR[91,2] = PR[90,2] + -6.297;
   1:L PR[91] R[100]mm/sec CNT100;
   1:  PR[91,1] = PR[90,1] + 8.267;
   1:  PR[91,2] = PR[90,2] + -8.216;
   1:L PR[91] R[100]mm/sec CNT100;
   1:  PR[91,1] = PR[90,1] + 9.033;
   1:  PR[91,2] = PR[90,2] + -9.857;
   1:L PR[91] R[100]mm/sec CNT100;
   1:  PR[91,1] = PR[90,1] + 10.075;
   1:  PR[91,2] = PR[90,2] + -11.344;
   1:L PR[91] R[100]mm/sec CNT100;
   1:  PR[91,1] = PR[90,1] + 11.336;
   1:  PR[91,2] = PR[90,2] + -12.985;
   1:L PR[91] R[100]mm/sec CNT100;
   1:  PR[91,1] = PR[90,1] + 12.591;
   1:  PR[91,2] = PR[90,2] + -14.240;
   1:L PR[91] R[100]mm/sec CNT100;
   1:  PR[91,1] = PR[90,1] + 14.216;
   1:  PR[91,2] = PR[90,2] + -15.482;
   1:L PR[91] R[100]mm/sec CNT100;
   1:  PR[91,1] = PR[90,1] + 15.723;
   1:  PR[91,2] = PR[90,2] + -16.536;
   1:L PR[91] R[100]mm/sec CNT100;
   1:  PR[91,1] = PR[90,1] + 17.382;
   1:  PR[91,2] = PR[90,2] + -17.310;
   1:L PR[91] R[100]mm/sec CNT100;
   1:  PR[91,1] = PR[90,1] + 19.260;
   1:  PR[91,2] = PR[90,2] + -18.084;
   1:L PR[91] R[100]mm/sec CNT100TB   .50sec,CALL END_PUD;
   1:  PR[92] = PR[91];
   1:  PR[92,3] = PR[92,3] + 20;
   1:J PR[92] 10% FINE;
   1:  PR[91,1] = PR[90,1] + 79.374;
   1:  PR[91,2] = PR[90,2] + -18.203;
   1:  PR[92] = PR[91];
   1:  PR[92,3] = PR[92,3] + 20;
   1:J PR[92] 10% FINE;
   1:L PR[91] R[100]mm/sec CNT100;
   1:  CALL LASER_DRAHT_START;
   1:  PR[91,1] = PR[90,1] + 81.810;
   1:  PR[91,2] = PR[90,2] + -17.342;
   1:L PR[91] R[100]mm/sec CNT100;
   1:  PR[91,1] = PR[90,1] + 82.898;
   1:  PR[91,2] = PR[90,2] + -16.835;
   1:L PR[91] R[100]mm/sec CNT100;
   1:  PR[91,1] = PR[90,1] + 84.947;
   1:  PR[91,2] = PR[90,2] + -15.539;
   1:L PR[91] R[100]mm/sec CNT100;
   1:  PR[91,1] = PR[90,1] + 86.009;
   1:  PR[91,2] = PR[90,2] + -14.796;
   1:L PR[91] R[100]mm/sec CNT100;
   1:  PR[91,1] = PR[90,1] + 88.630;
   1:  PR[91,2] = PR[90,2] + -12.166;
   1:L PR[91] R[100]mm/sec CNT100;
   1:  PR[91,1] = PR[90,1] + 89.414;
   1:  PR[91,2] = PR[90,2] + -11.047;
   1:L PR[91] R[100]mm/sec CNT100;
   1:  PR[91,1] = PR[90,1] + 90.618;
   1:  PR[91,2] = PR[90,2] + -9.123;
   1:L PR[91] R[100]mm/sec CNT100;
   1:  PR[91,1] = PR[90,1] + 91.216;
   1:  PR[91,2] = PR[90,2] + -7.842;
   1:L PR[91] R[100]mm/sec CNT100;
   1:  PR[91,1] = PR[90,1] + 91.941;
   1:  PR[91,2] = PR[90,2] + -5.760;
   1:L PR[91] R[100]mm/sec CNT100;
   1:  PR[91,1] = PR[90,1] + 92.309;
   1:  PR[91,2] = PR[90,2] + -4.387;
   1:L PR[91] R[100]mm/sec CNT100;
   1:  PR[91,1] = PR[90,1] + 92.441;
   1:  PR[91,2] = PR[90,2] + -2.880;
   1:L PR[91] R[100]mm/sec CNT100;
   1:  PR[91,1] = PR[90,1] + 92.682;
   1:  PR[91,2] = PR[90,2] + -0.706;
   1:L PR[91] R[100]mm/sec CNT100;
   1:  PR[91,1] = PR[90,1] + 92.553;
   1:  PR[91,2] = PR[90,2] + 0.769;
   1:L PR[91] R[100]mm/sec CNT100;
   1:  PR[91,1] = PR[90,1] + 92.315;
   1:  PR[91,2] = PR[90,2] + 2.905;
   1:L PR[91] R[100]mm/sec CNT100;
   1:  PR[91,1] = PR[90,1] + 91.941;
   1:  PR[91,2] = PR[90,2] + 4.301;
   1:L PR[91] R[100]mm/sec CNT100;
   1:  PR[91,1] = PR[90,1] + 91.216;
   1:  PR[91,2] = PR[90,2] + 6.383;
   1:L PR[91] R[100]mm/sec CNT100;
   1:  PR[91,1] = PR[90,1] + 90.619;
   1:  PR[91,2] = PR[90,2] + 7.663;
   1:L PR[91] R[100]mm/sec CNT100;
   1:  PR[91,1] = PR[90,1] + 89.415;
   1:  PR[91,2] = PR[90,2] + 9.586;
   1:L PR[91] R[100]mm/sec CNT100;
   1:  PR[91,1] = PR[90,1] + 88.631;
   1:  PR[91,2] = PR[90,2] + 10.706;
   1:L PR[91] R[100]mm/sec CNT100;
   1:  PR[91,1] = PR[90,1] + 86.011;
   1:  PR[91,2] = PR[90,2] + 13.335;
   1:L PR[91] R[100]mm/sec CNT100;
   1:  PR[91,1] = PR[90,1] + 84.950;
   1:  PR[91,2] = PR[90,2] + 14.079;
   1:L PR[91] R[100]mm/sec CNT100;
   1:  PR[91,1] = PR[90,1] + 82.901;
   1:  PR[91,2] = PR[90,2] + 15.375;
   1:L PR[91] R[100]mm/sec CNT100;
   1:  PR[91,1] = PR[90,1] + 81.814;
   1:  PR[91,2] = PR[90,2] + 15.882;
   1:L PR[91] R[100]mm/sec CNT100;
   1:  PR[91,1] = PR[90,1] + 79.377;
   1:  PR[91,2] = PR[90,2] + 16.743;
   1:L PR[91] R[100]mm/sec CNT100;
   1:  PR[91,1] = PR[90,1] + 78.351;
   1:  PR[91,2] = PR[90,2] + 17.019;
   1:L PR[91] R[100]mm/sec CNT100;
   1:  PR[91,1] = PR[90,1] + 77.186;
   1:  PR[91,2] = PR[90,2] + 17.121;
   1:L PR[91] R[100]mm/sec CNT100;
   1:  PR[91,1] = PR[90,1] + 74.553;
   1:  PR[91,2] = PR[90,2] + 17.433;
   1:L PR[91] R[100]mm/sec CNT100;
   1:  PR[91,1] = PR[90,1] + 73.600;
   1:  PR[91,2] = PR[90,2] + 17.350;
   1:L PR[91] R[100]mm/sec CNT100;
   1:  PR[91,1] = PR[90,1] + 70.750;
   1:  PR[91,2] = PR[90,2] + 17.041;
   1:L PR[91] R[100]mm/sec CNT100;
   1:  PR[91,1] = PR[90,1] + 69.967;
   1:  PR[91,2] = PR[90,2] + 16.832;
   1:L PR[91] R[100]mm/sec CNT100;
   1:  PR[91,1] = PR[90,1] + 67.027;
   1:  PR[91,2] = PR[90,2] + 15.817;
   1:L PR[91] R[100]mm/sec CNT100;
   1:  PR[91,1] = PR[90,1] + 66.438;
   1:  PR[91,2] = PR[90,2] + 15.543;
   1:L PR[91] R[100]mm/sec CNT100;
   1:  PR[91,1] = PR[90,1] + 63.580;
   1:  PR[91,2] = PR[90,2] + 13.763;
   1:L PR[91] R[100]mm/sec CNT100;
   1:  PR[91,1] = PR[90,1] + 63.178;
   1:  PR[91,2] = PR[90,2] + 13.481;
   1:L PR[91] R[100]mm/sec CNT100;
   1:  PR[91,1] = PR[90,1] + 60.340;
   1:  PR[91,2] = PR[90,2] + 10.664;
   1:L PR[91] R[100]mm/sec CNT100;
   1:  PR[91,1] = PR[90,1] + 60.145;
   1:  PR[91,2] = PR[90,2] + 10.386;
   1:L PR[91] R[100]mm/sec CNT100;
   1:  PR[91,1] = PR[90,1] + 58.173;
   1:  PR[91,2] = PR[90,2] + 7.267;
   1:L PR[91] R[100]mm/sec CNT100;
   1:  PR[91,1] = PR[90,1] + 58.083;
   1:  PR[91,2] = PR[90,2] + 7.075;
   1:L PR[91] R[100]mm/sec CNT100;
   1:  PR[91,1] = PR[90,1] + 56.803;
   1:  PR[91,2] = PR[90,2] + 3.434;
   1:L PR[91] R[100]mm/sec CNT100;
   1:  PR[91,1] = PR[90,1] + 56.769;
   1:  PR[91,2] = PR[90,2] + 3.311;
   1:L PR[91] R[100]mm/sec CNT100;
   1:  PR[91,1] = PR[90,1] + 56.322;
   1:  PR[91,2] = PR[90,2] + -0.729;
   1:L PR[91] R[100]mm/sec CNT100;
   1:  PR[91,1] = PR[90,1] + 56.769;
   1:  PR[91,2] = PR[90,2] + -4.770;
   1:L PR[91] R[100]mm/sec CNT100;
   1:  PR[91,1] = PR[90,1] + 56.803;
   1:  PR[91,2] = PR[90,2] + -4.893;
   1:L PR[91] R[100]mm/sec CNT100;
   1:  PR[91,1] = PR[90,1] + 58.083;
   1:  PR[91,2] = PR[90,2] + -8.533;
   1:L PR[91] R[100]mm/sec CNT100;
   1:  PR[91,1] = PR[90,1] + 58.172;
   1:  PR[91,2] = PR[90,2] + -8.726;
   1:L PR[91] R[100]mm/sec CNT100;
   1:  PR[91,1] = PR[90,1] + 60.145;
   1:  PR[91,2] = PR[90,2] + -11.845;
   1:L PR[91] R[100]mm/sec CNT100;
   1:  PR[91,1] = PR[90,1] + 60.340;
   1:  PR[91,2] = PR[90,2] + -12.122;
   1:L PR[91] R[100]mm/sec CNT100;
   1:  PR[91,1] = PR[90,1] + 63.177;
   1:  PR[91,2] = PR[90,2] + -14.940;
   1:L PR[91] R[100]mm/sec CNT100;
   1:  PR[91,1] = PR[90,1] + 63.579;
   1:  PR[91,2] = PR[90,2] + -15.221;
   1:L PR[91] R[100]mm/sec CNT100;
   1:  PR[91,1] = PR[90,1] + 66.436;
   1:  PR[91,2] = PR[90,2] + -17.001;
   1:L PR[91] R[100]mm/sec CNT100;
   1:  PR[91,1] = PR[90,1] + 67.025;
   1:  PR[91,2] = PR[90,2] + -17.275;
   1:L PR[91] R[100]mm/sec CNT100;
   1:  PR[91,1] = PR[90,1] + 69.964;
   1:  PR[91,2] = PR[90,2] + -18.289;
   1:L PR[91] R[100]mm/sec CNT100;
   1:  PR[91,1] = PR[90,1] + 70.727;
   1:  PR[91,2] = PR[90,2] + -18.494;
   1:L PR[91] R[100]mm/sec CNT100;
   1:  PR[91,1] = PR[90,1] + 71.603;
   1:  PR[91,2] = PR[90,2] + -18.571;
   1:L PR[91] R[100]mm/sec CNT100;
   1:  PR[91,1] = PR[90,1] + 74.600;
   1:  PR[91,2] = PR[90,2] + -18.893;
   1:L PR[91] R[100]mm/sec CNT100;
   1:  PR[91,1] = PR[90,1] + 75.555;
   1:  PR[91,2] = PR[90,2] + -18.810;
   1:L PR[91] R[100]mm/sec CNT100;
   1:  PR[91,1] = PR[90,1] + 78.319;
   1:  PR[91,2] = PR[90,2] + -18.486;
   1:L PR[91] R[100]mm/sec CNT100;
   1:  PR[91,1] = PR[90,1] + 79.374;
   1:  PR[91,2] = PR[90,2] + -18.203;
   1:L PR[91] R[100]mm/sec CNT100TB   .50sec,CALL END_PUD;
   1:  PR[92] = PR[91];
   1:  PR[92,3] = PR[92,3] + 20;
   1:J PR[92] 10% FINE;
   1:  PR[91,1] = PR[90,1] + -13.324;
   1:  PR[91,2] = PR[90,2] + -14.811;
   1:  PR[92] = PR[91];
   1:  PR[92,3] = PR[92,3] + 20;
   1:J PR[92] 10% FINE;
   1:L PR[91] R[100]mm/sec CNT100;
   1:  CALL LASER_DRAHT_START;
   1:  PR[91,1] = PR[90,1] + -10.690;
   1:  PR[91,2] = PR[90,2] + -12.186;
   1:L PR[91] R[100]mm/sec CNT100;
   1:  PR[91,1] = PR[90,1] + -9.931;
   1:  PR[91,2] = PR[90,2] + -11.102;
   1:L PR[91] R[100]mm/sec CNT100;
   1:  PR[91,1] = PR[90,1] + -8.665;
   1:  PR[91,2] = PR[90,2] + -9.095;
   1:L PR[91] R[100]mm/sec CNT100;
   1:  PR[91,1] = PR[90,1] + -8.124;
   1:  PR[91,2] = PR[90,2] + -7.935;
   1:L PR[91] R[100]mm/sec CNT100;
   1:  PR[91,1] = PR[90,1] + -7.319;
   1:  PR[91,2] = PR[90,2] + -5.641;
   1:L PR[91] R[100]mm/sec CNT100;
   1:  PR[91,1] = PR[90,1] + -7.002;
   1:  PR[91,2] = PR[90,2] + -4.457;
   1:L PR[91] R[100]mm/sec CNT100;
   1:  PR[91,1] = PR[90,1] + -6.887;
   1:  PR[91,2] = PR[90,2] + -3.146;
   1:L PR[91] R[100]mm/sec CNT100;
   1:  PR[91,1] = PR[90,1] + -6.634;
   1:  PR[91,2] = PR[90,2] + -0.713;
   1:L PR[91] R[100]mm/sec CNT100;
   1:  PR[91,1] = PR[90,1] + -6.754;
   1:  PR[91,2] = PR[90,2] + 0.661;
   1:L PR[91] R[100]mm/sec CNT100;
   1:  PR[91,1] = PR[90,1] + -6.743;
   1:  PR[91,2] = PR[90,2] + 0.745;
   1:L PR[91] R[100]mm/sec CNT100;
   1:  PR[91,1] = PR[90,1] + -6.995;
   1:  PR[91,2] = PR[90,2] + 2.973;
   1:L PR[91] R[100]mm/sec CNT100;
   1:  PR[91,1] = PR[90,1] + -7.318;
   1:  PR[91,2] = PR[90,2] + 4.181;
   1:L PR[91] R[100]mm/sec CNT100;
   1:  PR[91,1] = PR[90,1] + -8.124;
   1:  PR[91,2] = PR[90,2] + 6.476;
   1:L PR[91] R[100]mm/sec CNT100;
   1:  PR[91,1] = PR[90,1] + -8.664;
   1:  PR[91,2] = PR[90,2] + 7.636;
   1:L PR[91] R[100]mm/sec CNT100;
   1:  PR[91,1] = PR[90,1] + -9.931;
   1:  PR[91,2] = PR[90,2] + 9.643;
   1:L PR[91] R[100]mm/sec CNT100;
   1:  PR[91,1] = PR[90,1] + -10.690;
   1:  PR[91,2] = PR[90,2] + 10.727;
   1:L PR[91] R[100]mm/sec CNT100;
   1:  PR[91,1] = PR[90,1] + -13.324;
   1:  PR[91,2] = PR[90,2] + 13.352;
   1:L PR[91] R[100]mm/sec CNT100;
   1:  PR[91,1] = PR[90,1] + -14.452;
   1:  PR[91,2] = PR[90,2] + 14.142;
   1:L PR[91] R[100]mm/sec CNT100;
   1:  PR[91,1] = PR[90,1] + -16.362;
   1:  PR[91,2] = PR[90,2] + 15.336;
   1:L PR[91] R[100]mm/sec CNT100;
   1:  PR[91,1] = PR[90,1] + -17.670;
   1:  PR[91,2] = PR[90,2] + 15.946;
   1:L PR[91] R[100]mm/sec CNT100;
   1:  PR[91,1] = PR[90,1] + -19.701;
   1:  PR[91,2] = PR[90,2] + 16.649;
   1:L PR[91] R[100]mm/sec CNT100;
   1:  PR[91,1] = PR[90,1] + -21.136;
   1:  PR[91,2] = PR[90,2] + 17.034;
   1:L PR[91] R[100]mm/sec CNT100;
   1:  PR[91,1] = PR[90,1] + -22.710;
   1:  PR[91,2] = PR[90,2] + 17.172;
   1:L PR[91] R[100]mm/sec CNT100;
   1:  PR[91,1] = PR[90,1] + -24.807;
   1:  PR[91,2] = PR[90,2] + 17.401;
   1:L PR[91] R[100]mm/sec CNT100;
   1:  PR[91,1] = PR[90,1] + -26.374;
   1:  PR[91,2] = PR[90,2] + 17.263;
   1:L PR[91] R[100]mm/sec CNT100;
   1:  PR[91,1] = PR[90,1] + -28.370;
   1:  PR[91,2] = PR[90,2] + 17.032;
   1:L PR[91] R[100]mm/sec CNT100;
   1:  PR[91,1] = PR[90,1] + -29.946;
   1:  PR[91,2] = PR[90,2] + 16.609;
   1:L PR[91] R[100]mm/sec CNT100;
   1:  PR[91,1] = PR[90,1] + -31.756;
   1:  PR[91,2] = PR[90,2] + 15.971;
   1:L PR[91] R[100]mm/sec CNT100;
   1:  PR[91,1] = PR[90,1] + -33.282;
   1:  PR[91,2] = PR[90,2] + 15.259;
   1:L PR[91] R[100]mm/sec CNT100;
   1:  PR[91,1] = PR[90,1] + -34.839;
   1:  PR[91,2] = PR[90,2] + 14.276;
   1:L PR[91] R[100]mm/sec CNT100;
   1:  PR[91,1] = PR[90,1] + -36.254;
   1:  PR[91,2] = PR[90,2] + 13.284;
   1:L PR[91] R[100]mm/sec CNT100;
   1:  PR[91,1] = PR[90,1] + -38.793;
   1:  PR[91,2] = PR[90,2] + 10.740;
   1:L PR[91] R[100]mm/sec CNT100;
   1:  PR[91,1] = PR[90,1] + -39.804;
   1:  PR[91,2] = PR[90,2] + 9.296;
   1:L PR[91] R[100]mm/sec CNT100;
   1:  PR[91,1] = PR[90,1] + -40.740;
   1:  PR[91,2] = PR[90,2] + 7.801;
   1:L PR[91] R[100]mm/sec CNT100;
   1:  PR[91,1] = PR[90,1] + -41.496;
   1:  PR[91,2] = PR[90,2] + 6.178;
   1:L PR[91] R[100]mm/sec CNT100;
   1:  PR[91,1] = PR[90,1] + -42.066;
   1:  PR[91,2] = PR[90,2] + 4.545;
   1:L PR[91] R[100]mm/sec CNT100;
   1:  PR[91,1] = PR[90,1] + -42.527;
   1:  PR[91,2] = PR[90,2] + 2.825;
   1:L PR[91] R[100]mm/sec CNT100;
   1:  PR[91,1] = PR[90,1] + -42.690;
   1:  PR[91,2] = PR[90,2] + 0.956;
   1:L PR[91] R[100]mm/sec CNT100;
   1:  PR[91,1] = PR[90,1] + -42.882;
   1:  PR[91,2] = PR[90,2] + -0.754;
   1:L PR[91] R[100]mm/sec CNT100;
   1:  PR[91,1] = PR[90,1] + -42.725;
   1:  PR[91,2] = PR[90,2] + -2.557;
   1:L PR[91] R[100]mm/sec CNT100;
   1:  PR[91,1] = PR[90,1] + -42.533;
   1:  PR[91,2] = PR[90,2] + -4.259;
   1:L PR[91] R[100]mm/sec CNT100;
   1:  PR[91,1] = PR[90,1] + -42.066;
   1:  PR[91,2] = PR[90,2] + -6.003;
   1:L PR[91] R[100]mm/sec CNT100;
   1:  PR[91,1] = PR[90,1] + -41.497;
   1:  PR[91,2] = PR[90,2] + -7.637;
   1:L PR[91] R[100]mm/sec CNT100;
   1:  PR[91,1] = PR[90,1] + -40.740;
   1:  PR[91,2] = PR[90,2] + -9.259;
   1:L PR[91] R[100]mm/sec CNT100;
   1:  PR[91,1] = PR[90,1] + -39.804;
   1:  PR[91,2] = PR[90,2] + -10.754;
   1:L PR[91] R[100]mm/sec CNT100;
   1:  PR[91,1] = PR[90,1] + -38.794;
   1:  PR[91,2] = PR[90,2] + -12.198;
   1:L PR[91] R[100]mm/sec CNT100;
   1:  PR[91,1] = PR[90,1] + -36.255;
   1:  PR[91,2] = PR[90,2] + -14.743;
   1:L PR[91] R[100]mm/sec CNT100;
   1:  PR[91,1] = PR[90,1] + -34.840;
   1:  PR[91,2] = PR[90,2] + -15.734;
   1:L PR[91] R[100]mm/sec CNT100;
   1:  PR[91,1] = PR[90,1] + -33.283;
   1:  PR[91,2] = PR[90,2] + -16.718;
   1:L PR[91] R[100]mm/sec CNT100;
   1:  PR[91,1] = PR[90,1] + -31.756;
   1:  PR[91,2] = PR[90,2] + -17.430;
   1:L PR[91] R[100]mm/sec CNT100;
   1:  PR[91,1] = PR[90,1] + -29.947;
   1:  PR[91,2] = PR[90,2] + -18.068;
   1:L PR[91] R[100]mm/sec CNT100;
   1:  PR[91,1] = PR[90,1] + -28.398;
   1:  PR[91,2] = PR[90,2] + -18.483;
   1:L PR[91] R[100]mm/sec CNT100;
   1:  PR[91,1] = PR[90,1] + -26.694;
   1:  PR[91,2] = PR[90,2] + -18.632;
   1:L PR[91] R[100]mm/sec CNT100;
   1:  PR[91,1] = PR[90,1] + -24.757;
   1:  PR[91,2] = PR[90,2] + -18.859;
   1:L PR[91] R[100]mm/sec CNT100;
   1:  PR[91,1] = PR[90,1] + -23.192;
   1:  PR[91,2] = PR[90,2] + -18.722;
   1:L PR[91] R[100]mm/sec CNT100;
   1:  PR[91,1] = PR[90,1] + -21.158;
   1:  PR[91,2] = PR[90,2] + -18.499;
   1:L PR[91] R[100]mm/sec CNT100;
   1:  PR[91,1] = PR[90,1] + -19.701;
   1:  PR[91,2] = PR[90,2] + -18.108;
   1:L PR[91] R[100]mm/sec CNT100;
   1:  PR[91,1] = PR[90,1] + -17.670;
   1:  PR[91,2] = PR[90,2] + -17.405;
   1:L PR[91] R[100]mm/sec CNT100;
   1:  PR[91,1] = PR[90,1] + -16.363;
   1:  PR[91,2] = PR[90,2] + -16.795;
   1:L PR[91] R[100]mm/sec CNT100;
   1:  PR[91,1] = PR[90,1] + -14.452;
   1:  PR[91,2] = PR[90,2] + -15.601;
   1:L PR[91] R[100]mm/sec CNT100;
   1:  PR[91,1] = PR[90,1] + -13.324;
   1:  PR[91,2] = PR[90,2] + -14.811;
   1:L PR[91] R[100]mm/sec CNT100TB   .50sec,CALL END_PUD;
   1:  PR[92] = PR[91];
   1:  PR[92,3] = PR[92,3] + 20;
   1:J PR[92] 10% FINE;
   1:  PR[91,1] = PR[90,1] + -92.440;
   1:  PR[91,2] = PR[90,2] + -4.177;
   1:  PR[92] = PR[91];
   1:  PR[92,3] = PR[92,3] + 20;
   1:J PR[92] 10% FINE;
   1:L PR[91] R[100]mm/sec CNT100;
   1:  CALL LASER_DRAHT_START;
   1:  PR[91,1] = PR[90,1] + -92.023;
   1:  PR[91,2] = PR[90,2] + -5.734;
   1:L PR[91] R[100]mm/sec CNT100;
   1:  PR[91,1] = PR[90,1] + -91.453;
   1:  PR[91,2] = PR[90,2] + -7.494;
   1:L PR[91] R[100]mm/sec CNT100;
   1:  PR[91,1] = PR[90,1] + -90.783;
   1:  PR[91,2] = PR[90,2] + -8.931;
   1:L PR[91] R[100]mm/sec CNT100;
   1:  PR[91,1] = PR[90,1] + -89.838;
   1:  PR[91,2] = PR[90,2] + -10.569;
   1:L PR[91] R[100]mm/sec CNT100;
   1:  PR[91,1] = PR[90,1] + -88.947;
   1:  PR[91,2] = PR[90,2] + -11.841;
   1:L PR[91] R[100]mm/sec CNT100;
   1:  PR[91,1] = PR[90,1] + -87.641;
   1:  PR[91,2] = PR[90,2] + -13.296;
   1:L PR[91] R[100]mm/sec CNT100;
   1:  PR[91,1] = PR[90,1] + -86.584;
   1:  PR[91,2] = PR[90,2] + -14.352;
   1:L PR[91] R[100]mm/sec CNT100;
   1:  PR[91,1] = PR[90,1] + -84.932;
   1:  PR[91,2] = PR[90,2] + -15.557;
   1:L PR[91] R[100]mm/sec CNT100;
   1:  PR[91,1] = PR[90,1] + -83.747;
   1:  PR[91,2] = PR[90,2] + -16.386;
   1:L PR[91] R[100]mm/sec CNT100;
   1:  PR[91,1] = PR[90,1] + -82.435;
   1:  PR[91,2] = PR[90,2] + -16.997;
   1:L PR[91] R[100]mm/sec CNT100;
   1:  PR[91,1] = PR[90,1] + -80.541;
   1:  PR[91,2] = PR[90,2] + -17.846;
   1:L PR[91] R[100]mm/sec CNT100;
   1:  PR[91,1] = PR[90,1] + -79.240;
   1:  PR[91,2] = PR[90,2] + -18.194;
   1:L PR[91] R[100]mm/sec CNT100;
   1:  PR[91,1] = PR[90,1] + -77.089;
   1:  PR[91,2] = PR[90,2] + -18.656;
   1:L PR[91] R[100]mm/sec CNT100;
   1:  PR[91,1] = PR[90,1] + -75.846;
   1:  PR[91,2] = PR[90,2] + -18.765;
   1:L PR[91] R[100]mm/sec CNT100;
   1:  PR[91,1] = PR[90,1] + -73.501;
   1:  PR[91,2] = PR[90,2] + -18.770;
   1:L PR[91] R[100]mm/sec CNT100;
   1:  PR[91,1] = PR[90,1] + -72.367;
   1:  PR[91,2] = PR[90,2] + -18.670;
   1:L PR[91] R[100]mm/sec CNT100;
   1:  PR[91,1] = PR[90,1] + -69.912;
   1:  PR[91,2] = PR[90,2] + -18.155;
   1:L PR[91] R[100]mm/sec CNT100;
   1:  PR[91,1] = PR[90,1] + -68.947;
   1:  PR[91,2] = PR[90,2] + -17.896;
   1:L PR[91] R[100]mm/sec CNT100;
   1:  PR[91,1] = PR[90,1] + -67.975;
   1:  PR[91,2] = PR[90,2] + -17.442;
   1:L PR[91] R[100]mm/sec CNT100;
   1:  PR[91,1] = PR[90,1] + -65.634;
   1:  PR[91,2] = PR[90,2] + -16.410;
   1:L PR[91] R[100]mm/sec CNT100;
   1:  PR[91,1] = PR[90,1] + -64.902;
   1:  PR[91,2] = PR[90,2] + -15.897;
   1:L PR[91] R[100]mm/sec CNT100;
   1:  PR[91,1] = PR[90,1] + -62.685;
   1:  PR[91,2] = PR[90,2] + -14.296;
   1:L PR[91] R[100]mm/sec CNT100;
   1:  PR[91,1] = PR[90,1] + -62.141;
   1:  PR[91,2] = PR[90,2] + -13.752;
   1:L PR[91] R[100]mm/sec CNT100;
   1:  PR[91,1] = PR[90,1] + -60.195;
   1:  PR[91,2] = PR[90,2] + -11.598;
   1:L PR[91] R[100]mm/sec CNT100;
   1:  PR[91,1] = PR[90,1] + -59.814;
   1:  PR[91,2] = PR[90,2] + -11.055;
   1:L PR[91] R[100]mm/sec CNT100;
   1:  PR[91,1] = PR[90,1] + -58.287;
   1:  PR[91,2] = PR[90,2] + -8.419;
   1:L PR[91] R[100]mm/sec CNT100;
   1:  PR[91,1] = PR[90,1] + -58.046;
   1:  PR[91,2] = PR[90,2] + -7.902;
   1:L PR[91] R[100]mm/sec CNT100;
   1:  PR[91,1] = PR[90,1] + -57.071;
   1:  PR[91,2] = PR[90,2] + -4.909;
   1:L PR[91] R[100]mm/sec CNT100;
   1:  PR[91,1] = PR[90,1] + -56.942;
   1:  PR[91,2] = PR[90,2] + -4.427;
   1:L PR[91] R[100]mm/sec CNT100;
   1:  PR[91,1] = PR[90,1] + -56.610;
   1:  PR[91,2] = PR[90,2] + -0.727;
   1:L PR[91] R[100]mm/sec CNT100;
   1:  PR[91,1] = PR[90,1] + -56.627;
   1:  PR[91,2] = PR[90,2] + -0.529;
   1:L PR[91] R[100]mm/sec CNT100;
   1:  PR[91,1] = PR[90,1] + -57.001;
   1:  PR[91,2] = PR[90,2] + 3.010;
   1:L PR[91] R[100]mm/sec CNT100;
   1:  PR[91,1] = PR[90,1] + -57.055;
   1:  PR[91,2] = PR[90,2] + 3.211;
   1:L PR[91] R[100]mm/sec CNT100;
   1:  PR[91,1] = PR[90,1] + -58.141;
   1:  PR[91,2] = PR[90,2] + 6.549;
   1:L PR[91] R[100]mm/sec CNT100;
   1:  PR[91,1] = PR[90,1] + -58.256;
   1:  PR[91,2] = PR[90,2] + 6.795;
   1:L PR[91] R[100]mm/sec CNT100;
   1:  PR[91,1] = PR[90,1] + -59.958;
   1:  PR[91,2] = PR[90,2] + 9.735;
   1:L PR[91] R[100]mm/sec CNT100;
   1:  PR[91,1] = PR[90,1] + -60.172;
   1:  PR[91,2] = PR[90,2] + 10.040;
   1:L PR[91] R[100]mm/sec CNT100;
   1:  PR[91,1] = PR[90,1] + -62.342;
   1:  PR[91,2] = PR[90,2] + 12.444;
   1:L PR[91] R[100]mm/sec CNT100;
   1:  PR[91,1] = PR[90,1] + -62.690;
   1:  PR[91,2] = PR[90,2] + 12.792;
   1:L PR[91] R[100]mm/sec CNT100;
   1:  PR[91,1] = PR[90,1] + -65.163;
   1:  PR[91,2] = PR[90,2] + 14.581;
   1:L PR[91] R[100]mm/sec CNT100;
   1:  PR[91,1] = PR[90,1] + -65.696;
   1:  PR[91,2] = PR[90,2] + 14.953;
   1:L PR[91] R[100]mm/sec CNT100;
   1:  PR[91,1] = PR[90,1] + -66.279;
   1:  PR[91,2] = PR[90,2] + 15.225;
   1:L PR[91] R[100]mm/sec CNT100;
   1:  PR[91,1] = PR[90,1] + -69.018;
   1:  PR[91,2] = PR[90,2] + 16.438;
   1:L PR[91] R[100]mm/sec CNT100;
   1:  PR[91,1] = PR[90,1] + -69.761;
   1:  PR[91,2] = PR[90,2] + 16.637;
   1:L PR[91] R[100]mm/sec CNT100;
   1:  PR[91,1] = PR[90,1] + -72.504;
   1:  PR[91,2] = PR[90,2] + 17.215;
   1:L PR[91] R[100]mm/sec CNT100;
   1:  PR[91,1] = PR[90,1] + -73.401;
   1:  PR[91,2] = PR[90,2] + 17.293;
   1:L PR[91] R[100]mm/sec CNT100;
   1:  PR[91,1] = PR[90,1] + -76.023;
   1:  PR[91,2] = PR[90,2] + 17.289;
   1:L PR[91] R[100]mm/sec CNT100;
   1:  PR[91,1] = PR[90,1] + -77.040;
   1:  PR[91,2] = PR[90,2] + 17.200;
   1:L PR[91] R[100]mm/sec CNT100;
   1:  PR[91,1] = PR[90,1] + -79.447;
   1:  PR[91,2] = PR[90,2] + 16.684;
   1:L PR[91] R[100]mm/sec CNT100;
   1:  PR[91,1] = PR[90,1] + -80.523;
   1:  PR[91,2] = PR[90,2] + 16.396;
   1:L PR[91] R[100]mm/sec CNT100;
   1:  PR[91,1] = PR[90,1] + -81.590;
   1:  PR[91,2] = PR[90,2] + 15.898;
   1:L PR[91] R[100]mm/sec CNT100;
   1:  PR[91,1] = PR[90,1] + -83.794;
   1:  PR[91,2] = PR[90,2] + 14.910;
   1:L PR[91] R[100]mm/sec CNT100;
   1:  PR[91,1] = PR[90,1] + -84.797;
   1:  PR[91,2] = PR[90,2] + 14.208;
   1:L PR[91] R[100]mm/sec CNT100;
   1:  PR[91,1] = PR[90,1] + -86.648;
   1:  PR[91,2] = PR[90,2] + 12.859;
   1:L PR[91] R[100]mm/sec CNT100;
   1:  PR[91,1] = PR[90,1] + -87.563;
   1:  PR[91,2] = PR[90,2] + 11.944;
   1:L PR[91] R[100]mm/sec CNT100;
   1:  PR[91,1] = PR[90,1] + -89.027;
   1:  PR[91,2] = PR[90,2] + 10.314;
   1:L PR[91] R[100]mm/sec CNT100;
   1:  PR[91,1] = PR[90,1] + -89.806;
   1:  PR[91,2] = PR[90,2] + 9.201;
   1:L PR[91] R[100]mm/sec CNT100;
   1:  PR[91,1] = PR[90,1] + -90.865;
   1:  PR[91,2] = PR[90,2] + 7.366;
   1:L PR[91] R[100]mm/sec CNT100;
   1:  PR[91,1] = PR[90,1] + -91.454;
   1:  PR[91,2] = PR[90,2] + 6.102;
   1:L PR[91] R[100]mm/sec CNT100;
   1:  PR[91,1] = PR[90,1] + -92.094;
   1:  PR[91,2] = PR[90,2] + 4.129;
   1:L PR[91] R[100]mm/sec CNT100;
   1:  PR[91,1] = PR[90,1] + -92.458;
   1:  PR[91,2] = PR[90,2] + 2.771;
   1:L PR[91] R[100]mm/sec CNT100;
   1:  PR[91,1] = PR[90,1] + -92.586;
   1:  PR[91,2] = PR[90,2] + 1.306;
   1:L PR[91] R[100]mm/sec CNT100;
   1:  PR[91,1] = PR[90,1] + -92.801;
   1:  PR[91,2] = PR[90,2] + -0.747;
   1:L PR[91] R[100]mm/sec CNT100;
   1:  PR[91,1] = PR[90,1] + -92.688;
   1:  PR[91,2] = PR[90,2] + -2.037;
   1:L PR[91] R[100]mm/sec CNT100;
   1:  PR[91,1] = PR[90,1] + -92.646;
   1:  PR[91,2] = PR[90,2] + -2.204;
   1:L PR[91] R[100]mm/sec CNT100;
   1:  PR[91,1] = PR[90,1] + -92.440;
   1:  PR[91,2] = PR[90,2] + -4.177;
   1:L PR[91] R[100]mm/sec CNT100TB   .50sec,CALL END_PUD;
   1:  PR[92] = PR[91];
   1:  PR[92,3] = PR[92,3] + 20;
   1:J PR[92] 10% FINE;
   1:  PR[91] = PR[90];
   1:  PR[91,1] = PR[90,1] + 42.652;
   1:  PR[91,2] = PR[90,2] + 3.230;
   1:  PR[91,3] = PR[90,3] + 15.795;
   1:  PR[92] = PR[91];
   1:  PR[92,3] = PR[92,3] + 20;
   1:J PR[92] 10% FINE;
   1:L PR[91] R[100]mm/sec CNT100;
   1:  CALL LASER_DRAHT_START;
   1:  PR[91,1] = PR[90,1] + 42.243;
   1:  PR[91,2] = PR[90,2] + 4.755;
   1:L PR[91] R[100]mm/sec CNT100;
   1:  PR[91,1] = PR[90,1] + 41.335;
   1:  PR[91,2] = PR[90,2] + 6.950;
   1:L PR[91] R[100]mm/sec CNT100;
   1:  PR[91,1] = PR[90,1] + 40.654;
   1:  PR[91,2] = PR[90,2] + 8.410;
   1:L PR[91] R[100]mm/sec CNT100;
   1:  PR[91,1] = PR[90,1] + 39.726;
   1:  PR[91,2] = PR[90,2] + 9.735;
   1:L PR[91] R[100]mm/sec CNT100;
   1:  PR[91,1] = PR[90,1] + 38.277;
   1:  PR[91,2] = PR[90,2] + 11.629;
   1:L PR[91] R[100]mm/sec CNT100;
   1:  PR[91,1] = PR[90,1] + 37.176;
   1:  PR[91,2] = PR[90,2] + 12.729;
   1:L PR[91] R[100]mm/sec CNT100;
   1:  PR[91,1] = PR[90,1] + 35.266;
   1:  PR[91,2] = PR[90,2] + 14.198;
   1:L PR[91] R[100]mm/sec CNT100;
   1:  PR[91,1] = PR[90,1] + 33.964;
   1:  PR[91,2] = PR[90,2] + 15.109;
   1:L PR[91] R[100]mm/sec CNT100;
   1:  PR[91,1] = PR[90,1] + 32.525;
   1:  PR[91,2] = PR[90,2] + 15.779;
   1:L PR[91] R[100]mm/sec CNT100;
   1:  PR[91,1] = PR[90,1] + 30.284;
   1:  PR[91,2] = PR[90,2] + 16.712;
   1:L PR[91] R[100]mm/sec CNT100;
   1:  PR[91,1] = PR[90,1] + 28.807;
   1:  PR[91,2] = PR[90,2] + 17.107;
   1:L PR[91] R[100]mm/sec CNT100;
   1:  PR[91,1] = PR[90,1] + 26.365;
   1:  PR[91,2] = PR[90,2] + 17.433;
   1:L PR[91] R[100]mm/sec CNT100;
   1:  PR[91,1] = PR[90,1] + 24.821;
   1:  PR[91,2] = PR[90,2] + 17.567;
   1:L PR[91] R[100]mm/sec CNT100;
   1:  PR[91,1] = PR[90,1] + 23.274;
   1:  PR[91,2] = PR[90,2] + 17.432;
   1:L PR[91] R[100]mm/sec CNT100;
   1:  PR[91,1] = PR[90,1] + 20.811;
   1:  PR[91,2] = PR[90,2] + 17.111;
   1:L PR[91] R[100]mm/sec CNT100;
   1:  PR[91,1] = PR[90,1] + 19.415;
   1:  PR[91,2] = PR[90,2] + 16.737;
   1:L PR[91] R[100]mm/sec CNT100;
   1:  PR[91,1] = PR[90,1] + 17.947;
   1:  PR[91,2] = PR[90,2] + 16.052;
   1:L PR[91] R[100]mm/sec CNT100;
   1:  PR[91,1] = PR[90,1] + 15.633;
   1:  PR[91,2] = PR[90,2] + 15.099;
   1:L PR[91] R[100]mm/sec CNT100;
   1:  PR[91,1] = PR[90,1] + 14.427;
   1:  PR[91,2] = PR[90,2] + 14.254;
   1:L PR[91] R[100]mm/sec CNT100;
   1:  PR[91,1] = PR[90,1] + 12.410;
   1:  PR[91,2] = PR[90,2] + 12.711;
   1:L PR[91] R[100]mm/sec CNT100;
   1:  PR[91,1] = PR[90,1] + 11.382;
   1:  PR[91,2] = PR[90,2] + 11.683;
   1:L PR[91] R[100]mm/sec CNT100;
   1:  PR[91,1] = PR[90,1] + 9.817;
   1:  PR[91,2] = PR[90,2] + 9.647;
   1:L PR[91] R[100]mm/sec CNT100;
   1:  PR[91,1] = PR[90,1] + 8.962;
   1:  PR[91,2] = PR[90,2] + 8.427;
   1:L PR[91] R[100]mm/sec CNT100;
   1:  PR[91,1] = PR[90,1] + 8.334;
   1:  PR[91,2] = PR[90,2] + 7.079;
   1:L PR[91] R[100]mm/sec CNT100;
   1:  PR[91,1] = PR[90,1] + 7.345;
   1:  PR[91,2] = PR[90,2] + 4.697;
   1:L PR[91] R[100]mm/sec CNT100;
   1:  PR[91,1] = PR[90,1] + 6.985;
   1:  PR[91,2] = PR[90,2] + 3.350;
   1:L PR[91] R[100]mm/sec CNT100;
   1:  PR[91,1] = PR[90,1] + 6.849;
   1:  PR[91,2] = PR[90,2] + 1.793;
   1:L PR[91] R[100]mm/sec CNT100;
   1:  PR[91,1] = PR[90,1] + 6.515;
   1:  PR[91,2] = PR[90,2] + -0.772;
   1:L PR[91] R[100]mm/sec CNT100;
   1:  PR[91,1] = PR[90,1] + 6.649;
   1:  PR[91,2] = PR[90,2] + -2.307;
   1:L PR[91] R[100]mm/sec CNT100;
   1:  PR[91,1] = PR[90,1] + 6.973;
   1:  PR[91,2] = PR[90,2] + -4.767;
   1:L PR[91] R[100]mm/sec CNT100;
   1:  PR[91,1] = PR[90,1] + 7.346;
   1:  PR[91,2] = PR[90,2] + -6.157;
   1:L PR[91] R[100]mm/sec CNT100;
   1:  PR[91,1] = PR[90,1] + 8.334;
   1:  PR[91,2] = PR[90,2] + -8.538;
   1:L PR[91] R[100]mm/sec CNT100;
   1:  PR[91,1] = PR[90,1] + 8.963;
   1:  PR[91,2] = PR[90,2] + -9.887;
   1:L PR[91] R[100]mm/sec CNT100;
   1:  PR[91,1] = PR[90,1] + 9.818;
   1:  PR[91,2] = PR[90,2] + -11.108;
   1:L PR[91] R[100]mm/sec CNT100;
   1:  PR[91,1] = PR[90,1] + 11.384;
   1:  PR[91,2] = PR[90,2] + -13.144;
   1:L PR[91] R[100]mm/sec CNT100;
   1:  PR[91,1] = PR[90,1] + 12.412;
   1:  PR[91,2] = PR[90,2] + -14.172;
   1:L PR[91] R[100]mm/sec CNT100;
   1:  PR[91,1] = PR[90,1] + 14.429;
   1:  PR[91,2] = PR[90,2] + -15.714;
   1:L PR[91] R[100]mm/sec CNT100;
   1:  PR[91,1] = PR[90,1] + 15.674;
   1:  PR[91,2] = PR[90,2] + -16.586;
   1:L PR[91] R[100]mm/sec CNT100;
   1:  PR[91,1] = PR[90,1] + 17.045;
   1:  PR[91,2] = PR[90,2] + -17.224;
   1:L PR[91] R[100]mm/sec CNT100;
   1:  PR[91,1] = PR[90,1] + 19.376;
   1:  PR[91,2] = PR[90,2] + -18.185;
   1:L PR[91] R[100]mm/sec CNT100;
   1:  PR[91,1] = PR[90,1] + 20.817;
   1:  PR[91,2] = PR[90,2] + -18.571;
   1:L PR[91] R[100]mm/sec CNT100;
   1:  PR[91,1] = PR[90,1] + 23.280;
   1:  PR[91,2] = PR[90,2] + -18.892;
   1:L PR[91] R[100]mm/sec CNT100;
   1:  PR[91,1] = PR[90,1] + 24.827;
   1:  PR[91,2] = PR[90,2] + -19.026;
   1:L PR[91] R[100]mm/sec CNT100;
   1:  PR[91,1] = PR[90,1] + 26.371;
   1:  PR[91,2] = PR[90,2] + -18.891;
   1:L PR[91] R[100]mm/sec CNT100;
   1:  PR[91,1] = PR[90,1] + 28.813;
   1:  PR[91,2] = PR[90,2] + -18.565;
   1:L PR[91] R[100]mm/sec CNT100;
   1:  PR[91,1] = PR[90,1] + 30.248;
   1:  PR[91,2] = PR[90,2] + -18.180;
   1:L PR[91] R[100]mm/sec CNT100;
   1:  PR[91,1] = PR[90,1] + 31.746;
   1:  PR[91,2] = PR[90,2] + -17.481;
   1:L PR[91] R[100]mm/sec CNT100;
   1:  PR[91,1] = PR[90,1] + 34.002;
   1:  PR[91,2] = PR[90,2] + -16.542;
   1:L PR[91] R[100]mm/sec CNT100;
   1:  PR[91,1] = PR[90,1] + 35.268;
   1:  PR[91,2] = PR[90,2] + -15.655;
   1:L PR[91] R[100]mm/sec CNT100;
   1:  PR[91,1] = PR[90,1] + 37.179;
   1:  PR[91,2] = PR[90,2] + -14.185;
   1:L PR[91] R[100]mm/sec CNT100;
   1:  PR[91,1] = PR[90,1] + 38.278;
   1:  PR[91,2] = PR[90,2] + -13.086;
   1:L PR[91] R[100]mm/sec CNT100;
   1:  PR[91,1] = PR[90,1] + 39.728;
   1:  PR[91,2] = PR[90,2] + -11.192;
   1:L PR[91] R[100]mm/sec CNT100;
   1:  PR[91,1] = PR[90,1] + 40.655;
   1:  PR[91,2] = PR[90,2] + -9.868;
   1:L PR[91] R[100]mm/sec CNT100;
   1:  PR[91,1] = PR[90,1] + 41.336;
   1:  PR[91,2] = PR[90,2] + -8.408;
   1:L PR[91] R[100]mm/sec CNT100;
   1:  PR[91,1] = PR[90,1] + 42.243;
   1:  PR[91,2] = PR[90,2] + -6.213;
   1:L PR[91] R[100]mm/sec CNT100;
   1:  PR[91,1] = PR[90,1] + 42.640;
   1:  PR[91,2] = PR[90,2] + -4.731;
   1:L PR[91] R[100]mm/sec CNT100;
   1:  PR[91,1] = PR[90,1] + 42.787;
   1:  PR[91,2] = PR[90,2] + -3.048;
   1:L PR[91] R[100]mm/sec CNT100;
   1:  PR[91,1] = PR[90,1] + 43.061;
   1:  PR[91,2] = PR[90,2] + -0.700;
   1:L PR[91] R[100]mm/sec CNT100;
   1:  PR[91,1] = PR[90,1] + 42.958;
   1:  PR[91,2] = PR[90,2] + 0.480;
   1:L PR[91] R[100]mm/sec CNT100;
   1:  PR[91,1] = PR[90,1] + 42.951;
   1:  PR[91,2] = PR[90,2] + 0.952;
   1:L PR[91] R[100]mm/sec CNT100;
   1:  PR[91,1] = PR[90,1] + 42.651;
   1:  PR[91,2] = PR[90,2] + 3.230;
   1:L PR[91] R[100]mm/sec CNT100TB   .50sec,CALL END_PUD;
   1:  PR[92] = PR[91];
   1:  PR[92,3] = PR[92,3] + 20;
   1:J PR[92] 10% FINE;
   1:  PR[91,1] = PR[90,1] + 81.989;
   1:  PR[91,2] = PR[90,2] + -17.269;
   1:  PR[92] = PR[91];
   1:  PR[92,3] = PR[92,3] + 20;
   1:J PR[92] 10% FINE;
   1:L PR[91] R[100]mm/sec CNT100;
   1:  CALL LASER_DRAHT_START;
   1:  PR[91,1] = PR[90,1] + 82.662;
   1:  PR[91,2] = PR[90,2] + -16.955;
   1:L PR[91] R[100]mm/sec CNT100;
   1:  PR[91,1] = PR[90,1] + 85.199;
   1:  PR[91,2] = PR[90,2] + -15.350;
   1:L PR[91] R[100]mm/sec CNT100;
   1:  PR[91,1] = PR[90,1] + 85.902;
   1:  PR[91,2] = PR[90,2] + -14.858;
   1:L PR[91] R[100]mm/sec CNT100;
   1:  PR[91,1] = PR[90,1] + 88.613;
   1:  PR[91,2] = PR[90,2] + -12.136;
   1:L PR[91] R[100]mm/sec CNT100;
   1:  PR[91,1] = PR[90,1] + 89.154;
   1:  PR[91,2] = PR[90,2] + -11.363;
   1:L PR[91] R[100]mm/sec CNT100;
   1:  PR[91,1] = PR[90,1] + 90.647;
   1:  PR[91,2] = PR[90,2] + -8.978;
   1:L PR[91] R[100]mm/sec CNT100;
   1:  PR[91,1] = PR[90,1] + 91.071;
   1:  PR[91,2] = PR[90,2] + -8.070;
   1:L PR[91] R[100]mm/sec CNT100;
   1:  PR[91,1] = PR[90,1] + 91.970;
   1:  PR[91,2] = PR[90,2] + -5.488;
   1:L PR[91] R[100]mm/sec CNT100;
   1:  PR[91,1] = PR[90,1] + 92.233;
   1:  PR[91,2] = PR[90,2] + -4.507;
   1:L PR[91] R[100]mm/sec CNT100;
   1:  PR[91,1] = PR[90,1] + 92.330;
   1:  PR[91,2] = PR[90,2] + -3.402;
   1:L PR[91] R[100]mm/sec CNT100;
   1:  PR[91,1] = PR[90,1] + 92.629;
   1:  PR[91,2] = PR[90,2] + -0.706;
   1:L PR[91] R[100]mm/sec CNT100;
   1:  PR[91,1] = PR[90,1] + 92.534;
   1:  PR[91,2] = PR[90,2] + 0.375;
   1:L PR[91] R[100]mm/sec CNT100;
   1:  PR[91,1] = PR[90,1] + 92.239;
   1:  PR[91,2] = PR[90,2] + 3.025;
   1:L PR[91] R[100]mm/sec CNT100;
   1:  PR[91,1] = PR[90,1] + 91.971;
   1:  PR[91,2] = PR[90,2] + 4.029;
   1:L PR[91] R[100]mm/sec CNT100;
   1:  PR[91,1] = PR[90,1] + 91.071;
   1:  PR[91,2] = PR[90,2] + 6.611;
   1:L PR[91] R[100]mm/sec CNT100;
   1:  PR[91,1] = PR[90,1] + 90.648;
   1:  PR[91,2] = PR[90,2] + 7.518;
   1:L PR[91] R[100]mm/sec CNT100;
   1:  PR[91,1] = PR[90,1] + 89.155;
   1:  PR[91,2] = PR[90,2] + 9.903;
   1:L PR[91] R[100]mm/sec CNT100;
   1:  PR[91,1] = PR[90,1] + 88.614;
   1:  PR[91,2] = PR[90,2] + 10.676;
   1:L PR[91] R[100]mm/sec CNT100;
   1:  PR[91,1] = PR[90,1] + 85.903;
   1:  PR[91,2] = PR[90,2] + 13.398;
   1:L PR[91] R[100]mm/sec CNT100;
   1:  PR[91,1] = PR[90,1] + 85.201;
   1:  PR[91,2] = PR[90,2] + 13.890;
   1:L PR[91] R[100]mm/sec CNT100;
   1:  PR[91,1] = PR[90,1] + 82.664;
   1:  PR[91,2] = PR[90,2] + 15.495;
   1:L PR[91] R[100]mm/sec CNT100;
   1:  PR[91,1] = PR[90,1] + 81.991;
   1:  PR[91,2] = PR[90,2] + 15.809;
   1:L PR[91] R[100]mm/sec CNT100;
   1:  PR[91,1] = PR[90,1] + 78.976;
   1:  PR[91,2] = PR[90,2] + 16.875;
   1:L PR[91] R[100]mm/sec CNT100;
   1:  PR[91,1] = PR[90,1] + 78.416;
   1:  PR[91,2] = PR[90,2] + 17.025;
   1:L PR[91] R[100]mm/sec CNT100;
   1:  PR[91,1] = PR[90,1] + 77.732;
   1:  PR[91,2] = PR[90,2] + 17.085;
   1:L PR[91] R[100]mm/sec CNT100;
   1:  PR[91,1] = PR[90,1] + 74.475;
   1:  PR[91,2] = PR[90,2] + 17.471;
   1:L PR[91] R[100]mm/sec CNT100;
   1:  PR[91,1] = PR[90,1] + 74.032;
   1:  PR[91,2] = PR[90,2] + 17.433;
   1:L PR[91] R[100]mm/sec CNT100;
   1:  PR[91,1] = PR[90,1] + 70.510;
   1:  PR[91,2] = PR[90,2] + 17.051;
   1:L PR[91] R[100]mm/sec CNT100;
   1:  PR[91,1] = PR[90,1] + 70.253;
   1:  PR[91,2] = PR[90,2] + 16.983;
   1:L PR[91] R[100]mm/sec CNT100;
   1:  PR[91,1] = PR[90,1] + 66.623;
   1:  PR[91,2] = PR[90,2] + 15.730;
   1:L PR[91] R[100]mm/sec CNT100;
   1:  PR[91,1] = PR[90,1] + 66.560;
   1:  PR[91,2] = PR[90,2] + 15.701;
   1:L PR[91] R[100]mm/sec CNT100;
   1:  PR[91,1] = PR[90,1] + 63.099;
   1:  PR[91,2] = PR[90,2] + 13.539;
   1:L PR[91] R[100]mm/sec CNT100;
   1:  PR[91,1] = PR[90,1] + 61.504;
   1:  PR[91,2] = PR[90,2] + 11.958;
   1:L PR[91] R[100]mm/sec CNT100;
   1:  PR[91,1] = PR[90,1] + 60.153;
   1:  PR[91,2] = PR[90,2] + 10.655;
   1:L PR[91] R[100]mm/sec CNT100;
   1:  PR[91,1] = PR[90,1] + 57.910;
   1:  PR[91,2] = PR[90,2] + 7.206;
   1:L PR[91] R[100]mm/sec CNT100;
   1:  PR[91,1] = PR[90,1] + 56.513;
   1:  PR[91,2] = PR[90,2] + 3.344;
   1:L PR[91] R[100]mm/sec CNT100;
   1:  PR[91,1] = PR[90,1] + 56.084;
   1:  PR[91,2] = PR[90,2] + -0.301;
   1:L PR[91] R[100]mm/sec CNT100;
   1:  PR[91,1] = PR[90,1] + 56.083;
   1:  PR[91,2] = PR[90,2] + -0.618;
   1:L PR[91] R[100]mm/sec CNT100;
   1:  PR[91,1] = PR[90,1] + 56.222;
   1:  PR[91,2] = PR[90,2] + -1.824;
   1:L PR[91] R[100]mm/sec CNT100;
   1:  PR[91,1] = PR[90,1] + 56.519;
   1:  PR[91,2] = PR[90,2] + -4.820;
   1:L PR[91] R[100]mm/sec CNT100;
   1:  PR[91,1] = PR[90,1] + 57.910;
   1:  PR[91,2] = PR[90,2] + -8.665;
   1:L PR[91] R[100]mm/sec CNT100;
   1:  PR[91,1] = PR[90,1] + 60.153;
   1:  PR[91,2] = PR[90,2] + -12.114;
   1:L PR[91] R[100]mm/sec CNT100;
   1:  PR[91,1] = PR[90,1] + 61.504;
   1:  PR[91,2] = PR[90,2] + -13.416;
   1:L PR[91] R[100]mm/sec CNT100;
   1:  PR[91,1] = PR[90,1] + 63.099;
   1:  PR[91,2] = PR[90,2] + -14.998;
   1:L PR[91] R[100]mm/sec CNT100;
   1:  PR[91,1] = PR[90,1] + 66.560;
   1:  PR[91,2] = PR[90,2] + -17.159;
   1:L PR[91] R[100]mm/sec CNT100;
   1:  PR[91,1] = PR[90,1] + 66.622;
   1:  PR[91,2] = PR[90,2] + -17.188;
   1:L PR[91] R[100]mm/sec CNT100;
   1:  PR[91,1] = PR[90,1] + 70.252;
   1:  PR[91,2] = PR[90,2] + -18.441;
   1:L PR[91] R[100]mm/sec CNT100;
   1:  PR[91,1] = PR[90,1] + 70.505;
   1:  PR[91,2] = PR[90,2] + -18.509;
   1:L PR[91] R[100]mm/sec CNT100;
   1:  PR[91,1] = PR[90,1] + 74.521;
   1:  PR[91,2] = PR[90,2] + -18.931;
   1:L PR[91] R[100]mm/sec CNT100;
   1:  PR[91,1] = PR[90,1] + 74.969;
   1:  PR[91,2] = PR[90,2] + -18.892;
   1:L PR[91] R[100]mm/sec CNT100;
   1:  PR[91,1] = PR[90,1] + 78.386;
   1:  PR[91,2] = PR[90,2] + -18.492;
   1:L PR[91] R[100]mm/sec CNT100;
   1:  PR[91,1] = PR[90,1] + 78.974;
   1:  PR[91,2] = PR[90,2] + -18.335;
   1:L PR[91] R[100]mm/sec CNT100;
   1:  PR[91,1] = PR[90,1] + 81.989;
   1:  PR[91,2] = PR[90,2] + -17.269;
   1:L PR[91] R[100]mm/sec CNT100TB   .50sec,CALL END_PUD;
   1:  PR[92] = PR[91];
   1:  PR[92,3] = PR[92,3] + 20;
   1:J PR[92] 10% FINE;
   1:  PR[91,1] = PR[90,1] + -38.779;
   1:  PR[91,2] = PR[90,2] + 10.719;
   1:  PR[92] = PR[91];
   1:  PR[92,3] = PR[92,3] + 20;
   1:J PR[92] 10% FINE;
   1:L PR[91] R[100]mm/sec CNT100;
   1:  CALL LASER_DRAHT_START;
   1:  PR[91,1] = PR[90,1] + -39.599;
   1:  PR[91,2] = PR[90,2] + 9.548;
   1:L PR[91] R[100]mm/sec CNT100;
   1:  PR[91,1] = PR[90,1] + -40.764;
   1:  PR[91,2] = PR[90,2] + 7.688;
   1:L PR[91] R[100]mm/sec CNT100;
   1:  PR[91,1] = PR[90,1] + -41.382;
   1:  PR[91,2] = PR[90,2] + 6.362;
   1:L PR[91] R[100]mm/sec CNT100;
   1:  PR[91,1] = PR[90,1] + -42.091;
   1:  PR[91,2] = PR[90,2] + 4.328;
   1:L PR[91] R[100]mm/sec CNT100;
   1:  PR[91,1] = PR[90,1] + -42.468;
   1:  PR[91,2] = PR[90,2] + 2.922;
   1:L PR[91] R[100]mm/sec CNT100;
   1:  PR[91,1] = PR[90,1] + -42.603;
   1:  PR[91,2] = PR[90,2] + 1.375;
   1:L PR[91] R[100]mm/sec CNT100;
   1:  PR[91,1] = PR[90,1] + -42.842;
   1:  PR[91,2] = PR[90,2] + -0.754;
   1:L PR[91] R[100]mm/sec CNT100;
   1:  PR[91,1] = PR[90,1] + -42.713;
   1:  PR[91,2] = PR[90,2] + -2.236;
   1:L PR[91] R[100]mm/sec CNT100;
   1:  PR[91,1] = PR[90,1] + -42.474;
   1:  PR[91,2] = PR[90,2] + -4.356;
   1:L PR[91] R[100]mm/sec CNT100;
   1:  PR[91,1] = PR[90,1] + -42.092;
   1:  PR[91,2] = PR[90,2] + -5.786;
   1:L PR[91] R[100]mm/sec CNT100;
   1:  PR[91,1] = PR[90,1] + -41.382;
   1:  PR[91,2] = PR[90,2] + -7.820;
   1:L PR[91] R[100]mm/sec CNT100;
   1:  PR[91,1] = PR[90,1] + -40.765;
   1:  PR[91,2] = PR[90,2] + -9.146;
   1:L PR[91] R[100]mm/sec CNT100;
   1:  PR[91,1] = PR[90,1] + -39.599;
   1:  PR[91,2] = PR[90,2] + -11.006;
   1:L PR[91] R[100]mm/sec CNT100;
   1:  PR[91,1] = PR[90,1] + -38.780;
   1:  PR[91,2] = PR[90,2] + -12.177;
   1:L PR[91] R[100]mm/sec CNT100;
   1:  PR[91,1] = PR[90,1] + -36.170;
   1:  PR[91,2] = PR[90,2] + -14.794;
   1:L PR[91] R[100]mm/sec CNT100;
   1:  PR[91,1] = PR[90,1] + -35.034;
   1:  PR[91,2] = PR[90,2] + -15.590;
   1:L PR[91] R[100]mm/sec CNT100;
   1:  PR[91,1] = PR[90,1] + -33.098;
   1:  PR[91,2] = PR[90,2] + -16.813;
   1:L PR[91] R[100]mm/sec CNT100;
   1:  PR[91,1] = PR[90,1] + -31.890;
   1:  PR[91,2] = PR[90,2] + -17.377;
   1:L PR[91] R[100]mm/sec CNT100;
   1:  PR[91,1] = PR[90,1] + -29.641;
   1:  PR[91,2] = PR[90,2] + -18.169;
   1:L PR[91] R[100]mm/sec CNT100;
   1:  PR[91,1] = PR[90,1] + -28.443;
   1:  PR[91,2] = PR[90,2] + -18.491;
   1:L PR[91] R[100]mm/sec CNT100;
   1:  PR[91,1] = PR[90,1] + -27.100;
   1:  PR[91,2] = PR[90,2] + -18.608;
   1:L PR[91] R[100]mm/sec CNT100;
   1:  PR[91,1] = PR[90,1] + -24.694;
   1:  PR[91,2] = PR[90,2] + -18.890;
   1:L PR[91] R[100]mm/sec CNT100;
   1:  PR[91,1] = PR[90,1] + -23.504;
   1:  PR[91,2] = PR[90,2] + -18.786;
   1:L PR[91] R[100]mm/sec CNT100;
   1:  PR[91,1] = PR[90,1] + -20.978;
   1:  PR[91,2] = PR[90,2] + -18.509;
   1:L PR[91] R[100]mm/sec CNT100;
   1:  PR[91,1] = PR[90,1] + -19.899;
   1:  PR[91,2] = PR[90,2] + -18.219;
   1:L PR[91] R[100]mm/sec CNT100;
   1:  PR[91,1] = PR[90,1] + -17.379;
   1:  PR[91,2] = PR[90,2] + -17.346;
   1:L PR[91] R[100]mm/sec CNT100;
   1:  PR[91,1] = PR[90,1] + -16.438;
   1:  PR[91,2] = PR[90,2] + -16.908;
   1:L PR[91] R[100]mm/sec CNT100;
   1:  PR[91,1] = PR[90,1] + -14.070;
   1:  PR[91,2] = PR[90,2] + -15.428;
   1:L PR[91] R[100]mm/sec CNT100;
   1:  PR[91,1] = PR[90,1] + -13.284;
   1:  PR[91,2] = PR[90,2] + -14.878;
   1:L PR[91] R[100]mm/sec CNT100;
   1:  PR[91,1] = PR[90,1] + -10.558;
   1:  PR[91,2] = PR[90,2] + -12.163;
   1:L PR[91] R[100]mm/sec CNT100;
   1:  PR[91,1] = PR[90,1] + -10.046;
   1:  PR[91,2] = PR[90,2] + -11.432;
   1:L PR[91] R[100]mm/sec CNT100;
   1:  PR[91,1] = PR[90,1] + -8.477;
   1:  PR[91,2] = PR[90,2] + -8.945;
   1:L PR[91] R[100]mm/sec CNT100;
   1:  PR[91,1] = PR[90,1] + -8.123;
   1:  PR[91,2] = PR[90,2] + -8.185;
   1:L PR[91] R[100]mm/sec CNT100;
   1:  PR[91,1] = PR[90,1] + -7.125;
   1:  PR[91,2] = PR[90,2] + -5.344;
   1:L PR[91] R[100]mm/sec CNT100;
   1:  PR[91,1] = PR[90,1] + -6.924;
   1:  PR[91,2] = PR[90,2] + -4.592;
   1:L PR[91] R[100]mm/sec CNT100;
   1:  PR[91,1] = PR[90,1] + -6.848;
   1:  PR[91,2] = PR[90,2] + -3.726;
   1:L PR[91] R[100]mm/sec CNT100;
   1:  PR[91,1] = PR[90,1] + -6.535;
   1:  PR[91,2] = PR[90,2] + -0.713;
   1:L PR[91] R[100]mm/sec CNT100;
   1:  PR[91,1] = PR[90,1] + -6.614;
   1:  PR[91,2] = PR[90,2] + 0.189;
   1:L PR[91] R[100]mm/sec CNT100;
   1:  PR[91,1] = PR[90,1] + -6.599;
   1:  PR[91,2] = PR[90,2] + 0.298;
   1:L PR[91] R[100]mm/sec CNT100;
   1:  PR[91,1] = PR[90,1] + -6.917;
   1:  PR[91,2] = PR[90,2] + 3.108;
   1:L PR[91] R[100]mm/sec CNT100;
   1:  PR[91,1] = PR[90,1] + -7.125;
   1:  PR[91,2] = PR[90,2] + 3.885;
   1:L PR[91] R[100]mm/sec CNT100;
   1:  PR[91,1] = PR[90,1] + -8.123;
   1:  PR[91,2] = PR[90,2] + 6.726;
   1:L PR[91] R[100]mm/sec CNT100;
   1:  PR[91,1] = PR[90,1] + -8.477;
   1:  PR[91,2] = PR[90,2] + 7.486;
   1:L PR[91] R[100]mm/sec CNT100;
   1:  PR[91,1] = PR[90,1] + -10.046;
   1:  PR[91,2] = PR[90,2] + 9.972;
   1:L PR[91] R[100]mm/sec CNT100;
   1:  PR[91,1] = PR[90,1] + -10.557;
   1:  PR[91,2] = PR[90,2] + 10.703;
   1:L PR[91] R[100]mm/sec CNT100;
   1:  PR[91,1] = PR[90,1] + -13.284;
   1:  PR[91,2] = PR[90,2] + 13.419;
   1:L PR[91] R[100]mm/sec CNT100;
   1:  PR[91,1] = PR[90,1] + -14.070;
   1:  PR[91,2] = PR[90,2] + 13.969;
   1:L PR[91] R[100]mm/sec CNT100;
   1:  PR[91,1] = PR[90,1] + -16.438;
   1:  PR[91,2] = PR[90,2] + 15.449;
   1:L PR[91] R[100]mm/sec CNT100;
   1:  PR[91,1] = PR[90,1] + -17.378;
   1:  PR[91,2] = PR[90,2] + 15.887;
   1:L PR[91] R[100]mm/sec CNT100;
   1:  PR[91,1] = PR[90,1] + -19.898;
